# B&R Automation Studio project NAEUL004C00R13L518F00 (part 58)

#### Act_Background_TCPClose.st - Do Not Change!!!
```iecst
(** 2019-06-10 **)
ACTION Act_Background_TCPClose:

	//Close TCP Connection
	fbClose.udiTCPIdent	:= udiTCPIdent;
	fbClose(bEn := TRUE);

	IF fbClose.udiStatus = 0 THEN
		udiTCPIdent	:= 0;
		fbClose(bEn := FALSE);

		bRstConnection	:= FALSE;

	ELSIF fbClose.udiStatus < 65534 THEN
		udiTCPIdent	:= 0;
		eStatus1	:= Error;

		IF fbClose.udiStatus = 2300 THEN
			udiStatus1	:= 10027;	//Invalid Ident While Closing TCP
		ELSIF fbClose.udiStatus = 2310 THEN
			udiStatus1	:= 10028;	//Closing TCP Error
		ELSE
			udiStatus1	:= fbClose.udiStatus;
		END_IF

	END_IF

END_ACTION
```

#### Act_Background_Stop.st - Do Not Change!!!
```iecst
(** 2019-03-15 **)
ACTION Act_Background_Stop:

	IF bStop = TRUE THEN

		IF a_sMsgSend[0] = '' THEN

			bRstConnection	:= TRUE;

			IF udiTCPIdent = 0 THEN

				bRun	:= FALSE;

			END_IF

		END_IF

	END_IF

END_ACTION
```

#### Act_TCPSvr.st
```iecst
ACTION Act_TCPSvr:

	CASE usiStep OF
		0:
			//Analyse Connection
			IF udiSvrIdent = 0 THEN

				IF p_sSvrIP <> '' AND p_uiSvrPort <> 0 THEN
					usiStep	:= 1;
				END_IF

			ELSIF udiTCPIdent = 0 THEN

				usiStep	:= 2;

			END_IF

		1:
			//Create Server
			fbTCPSvrCreateSvr.sSvrIP				:= p_sSvrIP;
			fbTCPSvrCreateSvr.uiSvrPort				:= p_uiSvrPort;
			fbTCPSvrCreateSvr.udiAliveIdleTmInSec	:= 1;
			fbTCPSvrCreateSvr(bEn := TRUE);

			IF fbTCPSvrCreateSvr.udiStatus = 0 THEN
				udiSvrIdent	:= fbTCPSvrCreateSvr.udiTCPIdent;
				fbTCPSvrCreateSvr(bEn := FALSE);

				usiStep	:= 2;

			ELSIF fbTCPSvrCreateSvr.udiStatus < 65534 THEN
				fbTCPSvrCreateSvr(bEn := FALSE);

			END_IF

			IF p_bReconnect = TRUE THEN
				fbTCPSvrCreateSvr(bEn := FALSE);

				usiStep	:= 4;
			END_IF

		2:
			//Listen
			IF udiSvrIdent <> 0 THEN

				fbTCPSvrSvrListenFltr.bFltrIP			:= p_bFltrIP;
				fbTCPSvrSvrListenFltr.bFltrPort			:= p_bFltrPort;
				fbTCPSvrSvrListenFltr.a_sConfigIP[1]	:= p_sAllwClntIP;
				fbTCPSvrSvrListenFltr.a_uiConfigPort[1]	:= p_uiAllwClntPort;
				fbTCPSvrSvrListenFltr.udiSvrIdent		:= udiSvrIdent;
				fbTCPSvrSvrListenFltr(bEn := TRUE);

				IF fbTCPSvrSvrListenFltr.udiStatus = 0 THEN

					IF fbTCPSvrSvrListenFltr.bRejected = FALSE THEN
						udiTCPIdent	:= fbTCPSvrSvrListenFltr.udiClntIdent;
						fbTCPSvrSvrListenFltr(bEn := FALSE);
						bConnected		:= TRUE;

						usiStep	:= 3;
					ELSE
						fbTCPSvrSvrListenFltr(bEn := FALSE);
					END_IF

				ELSIF fbTCPSvrSvrListenFltr.udiStatus < 65534 THEN
					fbTCPSvrSvrListenFltr(bEn := FALSE);

				END_IF

			ELSE

				usiStep	:= 0;

			END_IF

			IF p_bReconnect = TRUE THEN
				fbTCPSvrSvrListenFltr(bEn := FALSE);

				usiStep	:= 4;
			END_IF

		3:
			//Send
			IF udiTCPIdent <> 0 AND bMsgSnd = TRUE THEN

				fbSend.udiTCPIdent	:= udiTCPIdent;
				fbSend.p_BffrDest	:= ADR(sMsgSnd);
				fbSend.udiSndSize	:= LEN(sMsgSnd);
				fbSend(bEn := TRUE);

				IF fbSend.udiStatus = 0 THEN
					bMsgSnd	:= FALSE;
					eSvrStat := SvrActIdle; //TCPSvrProcess
					fbSend(bEn := FALSE);

				ELSIF fbSend.udiStatus = 2320 THEN
					bMsgSnd	:= FALSE;
					fbSend(bEn := FALSE);

				ELSIF fbSend.udiStatus < 65534 THEN
					bMsgSnd	:= FALSE;
					fbSend(bEn := FALSE);

					usiStep	:= 4;

				END_IF

			ELSE
				fbSend(bEn := FALSE);

			END_IF

			//Receive
			IF udiTCPIdent <> 0 THEN

				fbRcv.udiTCPIdent	:= udiTCPIdent;
				fbRcv.p_BffrDest	:= ADR(sMsgRcv);
				fbRcv.udiBffrSize	:= SIZEOF(sMsgRcv);
				fbRcv(bEn := TRUE);

				IF eSvrStat <> SvrActWrite THEN
					eSvrStat := SvrActRead; //TCPSvrProcess
				END_IF

				IF fbRcv.udiStatus = 0 THEN
					bMsgRcv	:= TRUE;
					sSvrMsgRcv  := sMsgRcv;  //Evaluate
					fbRcv(bEn := FALSE);

				ELSIF fbRcv.udiStatus = 2316 THEN
					fbRcv(bEn := FALSE);

					usiStep	:= 4;

				ELSIF fbRcv.udiStatus = 2317 THEN //32605- no data is available for reading

					fbRcv(bEn := FALSE);
					memset(ADR(sMsgRcv) , 0 , SIZEOF(sMsgRcv));

				ELSIF fbRcv.udiStatus < 65534 THEN
					fbRcv(bEn := FALSE);

					usiStep	:= 4;

				END_IF

			ELSE
				fbRcv(bEn := FALSE);

			END_IF

			IF udiTCPIdent = 0 THEN
				usiStep	:= 0;
			END_IF

			IF p_bReconnect = TRUE THEN
				fbSend(bEn := FALSE);
				fbRcv(bEn := FALSE);

				usiStep	:= 4;
			END_IF

		4:
			//Close Client Ident
			IF udiTCPIdent <> 0 THEN

				fbClose.udiTCPIdent	:= udiTCPIdent;
				fbClose(bEn := TRUE);

				IF fbClose.udiStatus = 0 THEN
					udiTCPIdent	:= 0;
					fbClose(bEn := FALSE);
					bConnected		:= FALSE;

					usiStep	:= 5;

				ELSIF fbClose.udiStatus < 65534 THEN
					udiTCPIdent	:= 0;
					fbClose(bEn := FALSE);
					bConnected		:= FALSE;

				END_IF

			ELSE
				usiStep	:= 5;

			END_IF

		5:
			//Close Server Ident
			IF udiSvrIdent <> 0 THEN

				fbClose.udiTCPIdent	:= udiSvrIdent;
				fbClose(bEn := TRUE);

				IF fbClose.udiStatus = 0 THEN
					udiSvrIdent	:= 0;
					fbClose(bEn := FALSE);

					usiStep	:= 0;

				ELSIF fbClose.udiStatus < 65534 THEN
					udiSvrIdent	:= 0;
					fbClose(bEn := FALSE);

				END_IF

			ELSE
				usiStep	:= 0;

			END_IF

	END_CASE

END_ACTION
```

#### Act_TCPSvrProcess.st
```iecst
ACTION Act_TCPSvrProcess:

	CASE eSvrStat OF
		SvrActIdle:

		SvrActRead:
			//"Mag1Status","Mag2Status","Mag3Status","Mag4Status" >> 10:NA , 11:Error , 12:Ready, 13:Available ; 20:NA , 21:Error , 22:Ready, 23:Available

			eMagAGVStatus[0] := STRING_TO_USINT (LEFT(sSvrMsgRcv,FIND(sSvrMsgRcv, ',')-1));
			iSeparator 		:= FIND(sSvrMsgRcv, '$r$n');
			sData[0] := LEFT(sSvrMsgRcv, iSeparator-1);
			FOR i := 0 TO p_usiProjMag +(3 + 2*p_usiProjMag) DO 		//0:Dual ; 1:Triple; 2:Quar
				iSeparator := FIND(sData[i],',');
				IF iSeparator = 0 THEN
					;
				ELSE
					sData[i+1] := DELETE(sData[i],iSeparator+1,0);
				END_IF
			END_FOR

			IF bSingleMagLine THEN //single line magazine
				eMagAGVStatus[1] := STRING_TO_USINT (sData[1]);
			ELSE
				eMagAGVStatus[1] := STRING_TO_USINT (LEFT(sData[1],FIND(sData[1], ',')-1));
			END_IF

				eMagAGVStatus[2] := STRING_TO_USINT (LEFT(sData[2],FIND(sData[2], ',')-1));
			IF p_usiProjMag = 0 THEN//Dual mag
				eMagAGVStatus[3] := STRING_TO_USINT (sData[3]);
			ELSE //triple / quardrupal
				eMagAGVStatus[3] := STRING_TO_USINT (LEFT(sData[3],FIND(sData[3], ',')-1));
				eMagAGVStatus[4] := STRING_TO_USINT (LEFT(sData[4],FIND(sData[4], ',')-1));
				eMagAGVStatus[5] := STRING_TO_USINT (LEFT(sData[5],FIND(sData[5], ',')-1));
				eMagAGVStatus[6] := STRING_TO_USINT (LEFT(sData[6],FIND(sData[6], ',')-1));
				eMagAGVStatus[7] := STRING_TO_USINT (sData[7]);
			END_IF

			IF p_usiProjMag = 1 THEN//Triple mag
				eMagAGVStatus[5] := STRING_TO_USINT (sData[5]);
			ELSE
				eMagAGVStatus[5] := STRING_TO_USINT (LEFT(sData[5],FIND(sData[5], ',')-1));
				eMagAGVStatus[6] := STRING_TO_USINT (LEFT(sData[6],FIND(sData[6], ',')-1));
				eMagAGVStatus[7] := STRING_TO_USINT (sData[7]);
			END_IF

			IF eMagAGVStatus[0] >13 OR eMagAGVStatus[1] >12 OR eMagAGVStatus[2] >23 OR eMagAGVStatus[3] >22 OR
				eMagAGVStatus[4] >33 OR eMagAGVStatus[5] >32 OR eMagAGVStatus[6] >43 OR eMagAGVStatus[7] >42 OR

				eMagAGVStatus[0] <10 OR eMagAGVStatus[1] <10 OR eMagAGVStatus[2] <20 OR eMagAGVStatus[3] <20 OR
				eMagAGVStatus[4] <30 OR eMagAGVStatus[5] <30 OR eMagAGVStatus[6] <40 OR eMagAGVStatus[7] <40 THEN
				eSvrStatus := Error;
			END_IF

		SvrActRead1:
			//Structure: MagazineX, AGVStatus, AGVReq

			iSeparator 		:= FIND(sSvrMsgRcv, '$r$n');
			sData[0]		:= LEFT(sSvrMsgRcv, iSeparator-1); 		//magazine1 sData[0,1,2]
			sData[3] 		:= DELETE(sSvrMsgRcv,iSeparator+2,0);	//magazine2 sData[3,4,5]

			FOR i := 0 TO 5 DO
				iSeparator := FIND(sData[i],',');
				IF iSeparator = 0 THEN
					;
				ELSE
					sData[i+1] := DELETE(sData[i],iSeparator+1,0);
				END_IF
			END_FOR

			//check if endcode exist
			iSeparator := FIND(sData[i-1],'$r$n'); //where i = 6
			IF iSeparator = 0 THEN
				;
			ELSE
				sData[i-1] := DELETE(sData[i-1],iSeparator+1,iSeparator);
			END_IF

			tyAGVCurr[1].sAGVMag				:= LEFT(sData[0],FIND(sData[0], ',')-1);
			tyAGVCurr[1].eAGVStatus				:= STRING_TO_USINT (LEFT(sData[1],FIND(sData[1], ',')-1));
			tyAGVCurr[1].usiAGVReq				:= STRING_TO_USINT (sData[2]);
			tyAGVCurr[2].sAGVMag				:= LEFT(sData[3],FIND(sData[3], ',')-1);
			tyAGVCurr[2].eAGVStatus				:= STRING_TO_USINT (LEFT(sData[4],FIND(sData[4], ',')-1));
			tyAGVCurr[2].usiAGVReq				:= STRING_TO_USINT (sData[5]);

		SvrActWrite:
			//"Mag1Status","Mag2Status","Mag3Status","Mag4Status" >> 0:NA , 1:Error , 2:Ready, 3:Available
			//array [0][1]US1DS1 ,[2][3]US2DS2 ,[4][5]US3DS3, [6][7]US4DS4
			IF tyDTMagToAGV.bCI1Rdy  THEN
				a_sMagMcStatus[0] := '12'; //Ready, USB
			ELSE
				a_sMagMcStatus[0] := '10'; //NA
			END_IF
			IF tyDTMagToAGV.bCI1MagazineFull THEN
				a_sMagMcStatus[1] := '13'; //Available, DBA
			ELSE
				a_sMagMcStatus[1] := '10'; //NA
			END_IF;

			IF tyDTMagToAGV.bCI2Rdy  THEN
				a_sMagMcStatus[2] := '22';
			ELSE
				a_sMagMcStatus[2] := '20';
			END_IF;
			IF tyDTMagToAGV.bCI2MagazineFull THEN
				a_sMagMcStatus[3] := '23';
			ELSE
				a_sMagMcStatus[3] := '20';
			END_IF;

			IF tyDTMagToAGV.bCI3Rdy  THEN
				a_sMagMcStatus[4] := '32';
			ELSE
				a_sMagMcStatus[4] := '30';
			END_IF;
			IF tyDTMagToAGV.bCI3MagazineFull THEN
				a_sMagMcStatus[5] := '33';
			ELSE
				a_sMagMcStatus[5] := '30';
			END_IF;

			IF tyDTMagToAGV.bCI4Rdy  THEN
				a_sMagMcStatus[6] := '42';
			ELSE
				a_sMagMcStatus[6] := '40';
			END_IF;
			IF tyDTMagToAGV.bCI4MagazineFull THEN
				a_sMagMcStatus[7] := '43';
			ELSE
				a_sMagMcStatus[7] := '40';
			END_IF;
			//	sMsgSnd := USINT_TO_STRING (a_sMagMcStatus[3]);
			IF p_usiProjMag = 0 AND bSingleMagLine = FALSE THEN
				sMsgSnd := CONCAT(CONCAT(CONCAT(CONCAT(a_sMagMcStatus[0],','),CONCAT(a_sMagMcStatus[1],',')),CONCAT(a_sMagMcStatus[2],',')),CONCAT(a_sMagMcStatus[3],'$r$n'));
				bMsgSnd := TRUE;
			ELSIF bSingleMagLine THEN
				sMsgSnd := CONCAT(CONCAT(a_sMagMcStatus[0],','),CONCAT(a_sMagMcStatus[1],'$r$n'));
				bMsgSnd := TRUE;
			ELSE
				sMsgSnd := CONCAT(CONCAT(CONCAT(CONCAT(a_sMagMcStatus[0],','),CONCAT(a_sMagMcStatus[1],',')),CONCAT(a_sMagMcStatus[2],',')),a_sMagMcStatus[3]);
				sMsgSnd := CONCAT(CONCAT(CONCAT(CONCAT(CONCAT(sMsgSnd,','),CONCAT(a_sMagMcStatus[4],',')),CONCAT(a_sMagMcStatus[5],',')),CONCAT(a_sMagMcStatus[6],',')),CONCAT(a_sMagMcStatus[7],'$r$n'));
				bMsgSnd := TRUE;
			END_IF

	END_CASE;

	//Parse
	//Input (AGV to TCP(machine))
	bUBA 	:= eMagAGVStatus[0] = 13;
	bUBA2 	:= eMagAGVStatus[2] = 23;
	bDSB	:= eMagAGVStatus[1] = 12;
	bDSB2	:= eMagAGVStatus[3] = 22;

	//Output (Machine Sig(SOT) to TCP(AGV))
	tyDTMagToAGV.bCI1Rdy 			:= p_bUSB;
	tyDTMagToAGV.bCI1MagazineFull 	:= p_bDBA;
	tyDTMagToAGV.bCI2Rdy 			:= p_bUSB2;
	tyDTMagToAGV.bCI2MagazineFull 	:= p_bDBA2;

	fbTrig(CLK := p_bUSB);
	fbTrig1(CLK := p_bDBA);
	fbTrig2(CLK := p_bUSB2);
	fbTrig3(CLK := p_bDBA2);
	//	IF EDGEPOS(p_bUSB) OR EDGEPOS(p_bDBA) OR EDGEPOS(p_bUSB2) OR EDGEPOS(p_bDBA2)THEN
	IF fbTrig.Q OR fbTrig1.Q OR fbTrig2.Q OR fbTrig3.Q THEN
		eSvrStat := SvrActWrite;
	END_IF

END_ACTION
```

#### Act_Background_Log.st - Do Not Change!!!
```iecst
(** 2019-05-01 **)
ACTION Act_Background_Log:

	IF p_bLinkUIClearMsg THEN
		memset(ADR(a_tyHistoryList),0,SIZEOF(a_tyHistoryList));
		iHistoryCntr 	:= 1;
		p_bLinkUIClearMsg := FALSE;
	END_IF

	IF eStatus2 <> Error THEN

		IF udiWriteLogCntr <> udiLogCntr THEN

			CASE iWriteLogStep OF

				0:
					dtCurrDTTemp			:= p_dtCurrDT;
					fbFileAppend1.sFile		:= DT_TO_STRING(dtCurrDTTemp);
					fbFileAppend1.sFile		:= MID(fbFileAppend1.sFile , 10 , 4);
					fbFileAppend1.sFile		:= CONCAT('_' , fbFileAppend1.sFile);
					fbFileAppend1.sFile		:= CONCAT(p_sProgNm , fbFileAppend1.sFile);
					fbFileAppend1.sFile		:= CONCAT(fbFileAppend1.sFile , '.dat');

					fbFileAppend1.p_Src		:= ADR(a_sLogList[udiWriteLogCntr]);
					fbFileAppend1.udiLen	:= LEN(a_sLogList[udiWriteLogCntr]);

					iWriteLogStep	:= 1;

				1:
					fbFileAppend1(bEn := TRUE);
					IF fbFileAppend1.udiStatus = 0 THEN
						fbFileAppend1(bEn := FALSE);

						udiWriteLogCntr	:= udiWriteLogCntr + 1;
						IF udiWriteLogCntr = 11 THEN
							udiWriteLogCntr	:= 1;
						END_IF

						iWriteLogStep	:= 0;

					ELSIF fbFileAppend1.udiStatus < 65534 THEN
						eStatus2	:= Error;

						IF fbFileAppend1.udiStatus = 1900 THEN
							udiStatus2	:= 10018;	//File Open Error While Writing Log
						ELSIF fbFileAppend1.udiStatus = 1901 THEN
							udiStatus2	:= 10019;	//File Create Error While Writing Log
						ELSIF fbFileAppend1.udiStatus = 1913 THEN
							udiStatus2	:= 10020;	//Get File Info Error While Writing Log
						ELSIF fbFileAppend1.udiStatus = 1903 THEN
							udiStatus2	:= 10021;	//File Write Error While Writing Log
						ELSIF fbFileAppend1.udiStatus = 1904 THEN
							udiStatus2	:= 10022;	//File Close Error While Writing Log
						ELSIF fbFileAppend1.udiStatus = 1914 THEN
							udiStatus2	:= 10023;	//Directory Does Not Exist While Writing Log
						ELSE
							udiStatus2	:= fbFileAppend1.udiStatus;
						END_IF

						iWriteLogStep	:= 0;

					END_IF

			END_CASE

		END_IF

	END_IF

END_ACTION
```

#### Act_Main_Disable.st - Do Not Change!!!
```iecst
(** 2019-03-15 **)
ACTION Act_Main_Disable:

	bConnected		:= FALSE;

END_ACTION
```

#### InputRef.var - Do Not Change!!!
```iecst
(*2019-06-28*)
(**)
(*General*)
VAR
	p_bManual : REFERENCE TO BOOL;
	p_eAct : REFERENCE TO eTCPAction;
	p_udiRstErr : REFERENCE TO UDINT;
	p_bPrep : REFERENCE TO BOOL;
	p_bEn : REFERENCE TO BOOL;
	p_bDis : REFERENCE TO BOOL;
END_VAR
(**)
(*Configuration*)
VAR
	p_sSvrIP : REFERENCE TO STRING[15];
	p_uiSvrPort : REFERENCE TO UINT;
	p_uiClientPort : REFERENCE TO UINT;
	p_sMsgSnd : REFERENCE TO STRING[65535];
	p_sIPAddr : REFERENCE TO STRING[15];
	p_tyDTStructure : REFERENCE TO DTStructure;
	p_dtCurrDT : REFERENCE TO DATE_AND_TIME;
END_VAR
(*Listen Fltr*)
VAR
	p_eTCPModel : REFERENCE TO eTCPClientServer;
	p_bFltrIP : REFERENCE TO BOOL;
	p_bFltrPort : REFERENCE TO BOOL;
	p_sAllwClntIP : REFERENCE TO STRING[15];
	p_uiAllwClntPort : REFERENCE TO UINT;
	p_bReconnect : REFERENCE TO BOOL;
END_VAR
(**)
(*Input*)
VAR
	p_udiSndBffrSize : REFERENCE TO UDINT;
	p_udiRcvBffrSize : REFERENCE TO UDINT;
	p_udiAliveIdleTimeInSec : REFERENCE TO UDINT;
	p_tConnTimeOut : REFERENCE TO TIME;
	p_bOpsRun : REFERENCE TO BOOL;
	p_usiProjMag : REFERENCE TO USINT;
	p_sProgNm : REFERENCE TO STRING[15];
	p_bNtSettingsLoadDone : REFERENCE TO BOOL;
	p_udiFileKeepDay : REFERENCE TO UDINT;
END_VAR
(**)
VAR
	p_tyDTMagToAGV : REFERENCE TO tyTagDTMagToAGV;
END_VAR
(*Output from SOT to TCP*)
VAR
	p_bUSB : REFERENCE TO BOOL;
	p_bUSB2 : REFERENCE TO BOOL;
	p_bDBA : REFERENCE TO BOOL;
	p_bDBA2 : REFERENCE TO BOOL;
END_VAR
```

#### Act_Alarm.st - Do Not Change!!!
```iecst
(** 2019-03-25 **)
ACTION Act_Alarm:

	//Reset Error
	IF (eStatus = Error) AND bRstErr THEN
		p_eAct	:= TCPActIdle;
		eStat	:= TCPActIdle;
	END_IF

	IF p_udiRstErr <> udiRstErrOld THEN
		bRstErr			:= TRUE;
		udiRstErrOld	:= p_udiRstErr;
	ELSE
		bRstErr			:= FALSE;
	END_IF
	//Combine Error
	IF eStatus = Error OR eStatus1 = Error OR eStatus2 = Error THEN
		eMainStatus	:= Error;
	ELSE
		eMainStatus	:= eStatus;
	END_IF
	//Error
	IF EDGEPOS(eStatus = Error) THEN

		tyAlmData.sProgNm		:= p_sProgNm;
		tyAlmData.udiCode		:= udiStatus;
		tyAlmData.eSeverity		:= AlmSeverityError;
		tyAlmData.udiRunTime	:= tyAlmData.udiRunTime + 1;
		tyAlmData.bAlm			:= TRUE;
		tyAlmData.udiModuleNum  := udiModuleNum;
		g_sTCPProgNm		:= p_sProgNm;

		//Get Error Message
		IF tyAlmData.udiCode < 10000 OR tyAlmData.udiCode > 10199 THEN
			tyAlmData.sAlmMsg	:= 'Unknown';
			tyAlmData.sRcyMsg	:= 'Unknown';
		ELSE
			tyAlmData.sAlmMsg	:= a_tyAlmText[tyAlmData.udiCode].sAlmText;
			tyAlmData.sRcyMsg	:= a_tyAlmText[tyAlmData.udiCode].sRcyText;
		END_IF

		sStatTxt	:= tyAlmData.sAlmMsg;

	ELSIF bRstErr AND (tyAlmData.udiCode <> 0) THEN

		tyAlmData.udiCode	:= 0;
		tyAlmData.eSeverity	:= AlmSeverityNA;
		tyAlmData.sAlmMsg	:= '';
		tyAlmData.sRcyMsg	:= '';
		tyAlmData.bAlm			:= FALSE;
		sStatTxt	:= a_sStatText[eStat];

	END_IF

	//Error
	IF EDGEPOS(eStatus1 = Error) THEN

		tyAlmData1.sProgNm		:= p_sProgNm;
		tyAlmData1.udiCode		:= udiStatus1;
		tyAlmData1.eSeverity	:= AlmSeverityError;
		tyAlmData1.udiRunTime	:= tyAlmData1.udiRunTime + 1;
		tyAlmData1.bAlm			:= TRUE;
		tyAlmData1.udiModuleNum  := udiModuleNum;
		g_sTCPProgNm		:= p_sProgNm;

		//Get Error Message
		IF tyAlmData1.udiCode < 10000 OR tyAlmData1.udiCode > 10199 THEN
			tyAlmData1.sAlmMsg	:= 'Unknown';
			tyAlmData1.sRcyMsg	:= 'Unknown';
		ELSE
			tyAlmData1.sAlmMsg	:= a_tyAlmText[tyAlmData1.udiCode].sAlmText;
			tyAlmData1.sRcyMsg	:= a_tyAlmText[tyAlmData1.udiCode].sRcyText;
		END_IF

		sStatTxt	:= tyAlmData1.sAlmMsg;

	ELSIF bRstErr AND (tyAlmData1.udiCode <> 0) THEN

		tyAlmData1.udiCode		:= 0;
		tyAlmData1.eSeverity	:= AlmSeverityNA;
		tyAlmData1.sAlmMsg		:= '';
		tyAlmData1.sRcyMsg		:= '';
		tyAlmData1.bAlm			:= FALSE;
		sStatTxt	:= a_sStatText[eStat];

	END_IF

	//Error
	IF EDGEPOS(eStatus2 = Error) THEN

		tyAlmData2.sProgNm		:= p_sProgNm;
		tyAlmData2.udiCode		:= udiStatus2;
		tyAlmData2.eSeverity	:= AlmSeverityError;
		tyAlmData2.udiRunTime	:= tyAlmData2.udiRunTime + 1;
		tyAlmData2.bAlm			:= TRUE;
		tyAlmData2.udiModuleNum  := udiModuleNum;
		g_sTCPProgNm		:= p_sProgNm;

		//Get Error Message
		IF tyAlmData2.udiCode < 10000 OR tyAlmData2.udiCode > 10199 THEN
			tyAlmData2.sAlmMsg	:= 'Unknown';
			tyAlmData2.sRcyMsg	:= 'Unknown';
		ELSE
			tyAlmData2.sAlmMsg	:= a_tyAlmText[tyAlmData2.udiCode].sAlmText;
			tyAlmData2.sRcyMsg	:= a_tyAlmText[tyAlmData2.udiCode].sRcyText;
		END_IF

		sStatTxt	:= tyAlmData2.sAlmMsg;

	ELSIF bRstErr AND (tyAlmData2.udiCode <> 0) THEN

		tyAlmData2.udiCode		:= 0;
		tyAlmData2.eSeverity	:= AlmSeverityNA;
		tyAlmData2.sAlmMsg		:= '';
		tyAlmData2.sRcyMsg		:= '';
		tyAlmData2.bAlm			:= FALSE;
		sStatTxt	:= a_sStatText[eStat];

	END_IF

	//Error
	IF (bConnected = FALSE) THEN

		tyAlmData3.sProgNm		:= p_sProgNm;
		tyAlmData3.udiCode		:= udiStatus3;
		tyAlmData3.eSeverity	:= AlmSeverityWarning;
		tyAlmData3.udiRunTime	:= tyAlmData3.udiRunTime + 1;
		tyAlmData3.bWarning			:= TRUE;
		tyAlmData3.udiModuleNum  := udiModuleNum;
		g_sTCPProgNm		:= p_sProgNm;
		//Get Error Message
		IF tyAlmData3.udiCode < 10000 OR tyAlmData3.udiCode > 10199 THEN
			tyAlmData3.sAlmMsg	:= 'Unknown';
			tyAlmData3.sRcyMsg	:= 'Unknown';
		ELSE
			tyAlmData3.sAlmMsg	:= a_tyAlmText[tyAlmData3.udiCode].sAlmText;
			tyAlmData3.sRcyMsg	:= a_tyAlmText[tyAlmData3.udiCode].sRcyText;
			tyAlmData3.sRcyMsg	:= '';
		END_IF

		sStatTxt	:= tyAlmData3.sAlmMsg;

	ELSIF (bConnected AND (tyAlmData3.udiCode <> 0))  THEN

		tyAlmData3.udiCode		:= 0;
		tyAlmData3.eSeverity	:= AlmSeverityNA;
		tyAlmData3.sAlmMsg		:= '';
		tyAlmData3.sRcyMsg		:= '';
		tyAlmData3.bWarning		:= FALSE;
		sStatTxt	:= a_sStatText[eStat];

	END_IF
END_ACTION
```

#### Local.var - Do Not Change!!!
```iecst
(*2020-09-10*)
(**)
(*Local Action, State & Status*)
VAR
	bManual : BOOL := FALSE;
	eAct : eTCPAction := TCPActIdle;
	eStat : eTCPAction := TCPActIdle;
	eMainStatus : eFBStatus := Idle;
	eStatus : eFBStatus := Idle;
	eStatus1 : eFBStatus := Idle;
	eStatus2 : eFBStatus := Idle;
	udiStatus : UDINT := 0;
	udiStatus1 : UDINT := 0;
	udiStatus2 : UDINT := 0;
	udiStatus3 : UDINT := 0;
	udiStatus4 : UDINT := 0;
	udiStatus5 : UDINT := 0;
	sStatTxt : STRING[200] := '';
	a_sStatText : ARRAY[0..50] OF STRING[200] := ['Idling','Creating Directory','Deleting Old Log',48('')];
END_VAR
(**)
(*Local Alarm*)
VAR
	tyAlmData : tyAlmDat;
	tyAlmData1 : tyAlmDat;
	tyAlmData2 : tyAlmDat;
	tyAlmData3 : tyAlmDat;
	a_tyAlmText : ARRAY[10000..10199] OF tyAlmTxt := [(sAlmText:='Invalid Ident While Client Connecting',sRcyText:='Problem Occurred In The TCP/IP Connection. Check The Connection And Try To Reconnect.'),(sAlmText:='Setting Keep Alive Interval Time Error While Client Connecting',sRcyText:='Unable To Establish Connection Between Machine. Check For Setting And Resume Operation.'),(sAlmText:='Setting Keep Alive Idle Time Error While Client Connecting',sRcyText:='Unable To Establish Connection Between Machine. Check For Setting And Resume Operation.'),(sAlmText:='Setting Keep Alive Count Error While Client Connecting',sRcyText:='Unable To Establish Connection Between Machine. Check For Setting And Resume Operation.'),(sAlmText:='Setting Keep Alive Error While Client Connecting',sRcyText:='Unable To Establish Connection Between Machine. Check For Setting And Resume Operation.'),(sAlmText:='Setting Receive Buffer Error While Client Connecting',sRcyText:='Unable To Establish Connection Between Machine. Check For Setting And Resume Operation.'),(sAlmText:='Setting Send Buffer Error While Client Connecting',sRcyText:='Unable To Establish Connection Between Machine. Check For Setting And Resume Operation.'),(sAlmText:='Setting No Waiting Error While Client Connecting',sRcyText:='Unable To Establish Connection Between Machine. Check For Setting And Resume Operation.'),(sAlmText:='TCP Open Port Error While Client Connecting',sRcyText:='Problem Occurred In The TCP/IP Connection. Check The Connection And Try To Reconnect.'),(sAlmText:='Closing TCP Error While Client Connecting',sRcyText:='Problem Occurred In The TCP/IP Connection. Check The Connection And Try To Reconnect.'),(sAlmText:='Server Connection Failed While Client Connecting',sRcyText:='There Was A Problem Connecting To The Server. The Server May Not Exist or It is Unavailable At This Time. Check The Connection and Try Again.'),(sAlmText:='Ident In Used While Client Connecting',sRcyText:='Problem Occurred In The TCP/IP Connection. Check The Connection And Reconnect.'),(sAlmText:='TCP Connection Lost',sRcyText:='There Was A Problem Connecting To The Server. The Server May Not Exist or It is Unavailable At This Time. Check The Connection and Try Again.'),(sAlmText:='TCP Connection Lost',sRcyText:='Please Check Network Connection.'),(sAlmText:='Invalid Ident While Receiving Data',sRcyText:='Problem Occurred In The TCP/IP Connection. Check The Connection And Try To Reconnect.'),(sAlmText:='TCP Receive Data Error While Receiving Data',sRcyText:='Problem Occurred In The TCP/IP Connection. Check The Connection And Try To Reconnect.'),(sAlmText:='Create User Directory Error',sRcyText:='An Error Occurred While Attempting To Create User Directory. Please Contact Nutek For A Possible Solution'),(sAlmText:='Create Log Directory Error',sRcyText:='An Error Occurred While Attempting To Create User Directory. Please Contact Nutek For A Possible Solution'),(sAlmText:='File Open Error While Writing Log',sRcyText:='An Error Was Encountered While Trying To Open File. Please Contact Nutek For A Possible Solution.'),(sAlmText:='File Create Error While Writing Log',sRcyText:='An Error Was Encountered While Trying To Create File. Please Contact Nutek For A Possible Solution.'),(sAlmText:='Get File Info Error While Writing Log',sRcyText:='An Error Was Encountered While Getting File Info. Please Contact Nutek For A Possible Solution.'),(sAlmText:='File Write Error While Writing Log',sRcyText:='An Error Was Encountered While Getting File Info. Please Contact Nutek For A Possible Solution.'),(sAlmText:='File Close Error While Writing Log',sRcyText:='An Error Was Encountered While Trying To Close File. Please Contact Nutek For A Possible Solution.'),(sAlmText:='Directory Does Not Exist While Writing Log',sRcyText:='The Directory Does Not Exist.Please Contact Nutek For A Possible Solution.'),(sAlmText:='Invalid Ident While Sending Data',sRcyText:='Invalid Ident Value.'),(sAlmText:='TCP Retry Send Data Error While Sending Data',sRcyText:='Problem Occurred In The TCP/IP Connection. Check The Connection And Try To Reconnect.'),(sAlmText:='TCP Send Data Error',sRcyText:='Problem Occurred In The TCP/IP Connection. Check The Connection And Try To Reconnect.'),(sAlmText:='Invalid Ident While Closing TCP',sRcyText:='Invalid Ident Value.'),(sAlmText:='Closing TCP Error',sRcyText:='Problem Occurred In The TCP/IP Connection. Check The Connection And Try To Reconnect.'),171(0)];
END_VAR
(**)
(*Local Output*)
VAR
	bConnected : BOOL;
	bUSB : BOOL;
	bUBA : BOOL;
	bDSB : BOOL;
	bDBA : BOOL;
	bUSB2 : BOOL;
	bUBA2 : BOOL;
	bDSB2 : BOOL;
	bDBA2 : BOOL;
END_VAR
(**)
(*Local Input*)
VAR
	sSvrIP : STRING[15] := '192.168.0.16';
	uiSvrPort : UINT := 7171;
	uiClientPort : UINT := 5000;
	udiRstErr : UDINT := 0;
	bPrep : BOOL := TRUE;
	bEn : BOOL := TRUE;
	bDis : BOOL := FALSE;
	sIPAddr : STRING[15] := '192.168.0.16';
	tyDTStructure : DTStructure := (year:=2019,month:=01,day:=05,wday:=05,hour:=21,minute:=28,second:=30,millisec:=123,microsec:=456);
	dtCurrDT : DATE_AND_TIME := DT#2019-02-23-12:30:50;
	udiSndBffrSize : UDINT := 65536;
	udiRcvBffrSize : UDINT := 65536;
	udiAliveIdleTimeInSec : UDINT := 5;
	tConnTimeOut : TIME := T#30s;
	bOpsRun : BOOL := FALSE;
	udiFileKeepDay : UDINT := 30;
	usiProjMag : USINT := 0;
	sProgNm : STRING[15] := 'TCP';
	bNtSettingsLoadDone : BOOL := TRUE;
END_VAR
(**)
(*Local*)
VAR
	eTCPModel : eTCPClientServer := Server;
	eStatOld : eTCPAction := TCPActIdle;
	bRstErr : BOOL;
	udiRstErrOld : UDINT;
	bInitDone : BOOL;
	bInitialDone : BOOL;
	bRun : BOOL;
	bStop : BOOL;
	bRstConnection : BOOL;
	bRstState : BOOL;
	usiStep : USINT;
	udiTCPIdent : UDINT; (*Client ident*)
	udiMsgSendBffr : UDINT;
	udiSndMsgLen : UDINT;
	iFindBatteryLvl : INT;
	rCurrentBatteryLvl : REAL;
	sExtractBatteryLvl : STRING[30];
	sDecodeMsg : STRING[65535];
	a_sMsgSend : ARRAY[0..50] OF STRING[65535];
	bMsgSnd : BOOL;
	bMsgRcv : BOOL;
	sMsgSnd : STRING[65535];
	sMsgRcv : STRING[65535];
	sSvrMsgRcv : STRING[65535];
	sSnd : STRING[65535];
	sRcv : STRING[65535];
	fbClntConnect : fbTCPClntConnect;
	fbTCPSvrCreateSvr : fbTCPCreateSvr;
	fbTCPSvrSvrListenFltr : fbTCPSvrListenFltr;
	fbRcv : fbTCPRcv;
	fbSend : fbTCPSnd;
	fbClose : fbTCPClose;
	fbTrig : RF_TRIG;
	fbTrig1 : RF_TRIG;
	fbTrig2 : RF_TRIG;
	fbTrig3 : RF_TRIG;
	udiLogCntr : UDINT := 1;
	udiWriteLogCntr : UDINT := 1;
	a_sLogList : ARRAY[1..10] OF STRING[65535];
	sDT : STRING[80];
	dtCurrDTTemp : DATE_AND_TIME;
	fbDirCreate1 : fbDirCreate;
	fbDirCreate2 : fbDirCreate;
	fbFileAppend1 : fbFileFullAppend;
	fbFileOldDel1 : fbFileOldDel;
	iWriteLogStep : INT := 0;
	iHistoryCntr : INT := 1;
	a_tyHistoryList : ARRAY[1..8] OF tyTCPHistoryMsg;
	bLoginSuccess : BOOL;
	bCheckAliveTimeout : BOOL;
	bWaitAliveResponse : BOOL;
	fbSendAliveTimer : TON;
	fbCheckAliveTimer : TON;
END_VAR
(**)
VAR
	tyAIVMsgRcvData : tyAIVMsgRcvDat;
	sELD1Reached : STRING[80] := 'Arrived At ELD1';
	sELD1Completed : STRING[80] := 'ELD1_completed';
	sELD2Reached : STRING[80] := 'Arrived At ELD2';
	sELD2Completed : STRING[80] := 'ELD2_completed';
	sELD3Reached : STRING[80] := 'Arrived At ELD3';
	sELD3Completed : STRING[80] := 'ELD3_completed';
	sEUL1Reached : STRING[80] := 'Arrived At EUL1';
	sEUL1Completed : STRING[80] := 'EUL1_completed';
	sEUL2Reached : STRING[80] := 'Arrived At EUL2';
	sEUL2Completed : STRING[80] := 'EUL2_completed';
	sEUL3Reached : STRING[80] := 'Arrived At EUL3';
	sEUL3Completed : STRING[80] := 'EUL3_completed';
	sSTANDBYReached : STRING[80] := 'Arrived At STANDBY';
	sSTANDBYCompleted : STRING[80] := 'STANDBY_completed';
END_VAR
(*Server*)
VAR
	udiSvrIdent : UDINT := 0;
	bFltrIP : BOOL;
	bFltrPort : BOOL;
	sAllwClntIP : STRING[15];
	uiAllwClntPort : UINT;
	bReconnect : BOOL;
	eSvrStat : eTCPSvrAction := SvrActIdle;
	eSvrStatus : eFBStatus := Idle;
	bSingleMagLine : BOOL := FALSE;
END_VAR
(**)
(*Data Parameter(Read1)*)
VAR
	i : INT;
	iSeparator : INT := 0;
	tyAGVCurr : ARRAY[1..2] OF tyTCPAGVDetail;
	sData : ARRAY[0..7] OF STRING[30]; (*Buffer *)
END_VAR
(*Data Parameter(Read/write)*)
VAR
	eMagAGVStatus : ARRAY[0..7] OF eTCPAGVStatus := [8(AGVNA)];
	a_sMagMcStatus : ARRAY[0..7] OF STRING[2] := [8('')];
	tyDTMagToAGV : tyTagDTMagToAGV;
	udiModuleNum : UDINT := 4301;
END_VAR
```

#### Act_Action.st - not listed in the package file held
```iecst
(** 2019-03-25 **)
ACTION Act_Action:

//Reset Error
	IF (eStatus = Error) AND bRstErr THEN
		p_eAct	:= TCPActIdle;
		eStat	:= TCPActIdle;
	END_IF

	//Set p_eAct
	IF eStatus = Idle OR eStatus = Busy OR eStatus = Done THEN
		eStat	:= p_eAct;
	END_IF

END_ACTION
```

#### Act_Alarm1.st - not listed in the package file held
```iecst
(** 2019-03-25 **)
ACTION Act_Alarm1:

	//Error
	IF EDGEPOS(eStatus1 = Error) THEN

		tyAlmData1.sProgNm		:= p_sProgNm;
		tyAlmData1.udiCode		:= udiStatus1;
		tyAlmData1.eSeverity	:= AlmSeverityError;
		tyAlmData1.udiRunTime	:= tyAlmData1.udiRunTime + 1;
		tyAlmData1.bAlm			:= TRUE;
		tyAlmData1.udiModuleNum  := udiModuleNum;
		g_sTCPProgNm		:= p_sProgNm;

		//Get Error Message
		IF tyAlmData1.udiCode < 10000 OR tyAlmData1.udiCode > 10199 THEN
			tyAlmData1.sAlmMsg	:= 'Unknown';
			tyAlmData1.sRcyMsg	:= 'Unknown';
		ELSE
			tyAlmData1.sAlmMsg	:= a_tyAlmText[tyAlmData1.udiCode].sAlmText;
			tyAlmData1.sRcyMsg	:= a_tyAlmText[tyAlmData1.udiCode].sRcyText;
		END_IF

		sStatTxt	:= tyAlmData1.sAlmMsg;

	ELSIF bRstErr AND (tyAlmData1.udiCode <> 0) THEN

		tyAlmData1.udiCode		:= 0;
		tyAlmData1.eSeverity	:= AlmSeverityNA;
		tyAlmData1.sAlmMsg		:= '';
		tyAlmData1.sRcyMsg		:= '';
		tyAlmData1.bAlm			:= FALSE;
		sStatTxt	:= a_sStatText[eStat];

	END_IF

END_ACTION
```

#### Act_Alarm2.st - not listed in the package file held
```iecst
(** 2019-03-25 **)
ACTION Act_Alarm2:

	//Error
	IF EDGEPOS(eStatus2 = Error) THEN

		tyAlmData2.sProgNm		:= p_sProgNm;
		tyAlmData2.udiCode		:= udiStatus2;
		tyAlmData2.eSeverity	:= AlmSeverityError;
		tyAlmData2.udiRunTime	:= tyAlmData2.udiRunTime + 1;
		tyAlmData2.bAlm			:= TRUE;
		tyAlmData2.udiModuleNum  := udiModuleNum;
		g_sTCPProgNm		:= p_sProgNm;

		//Get Error Message
		IF tyAlmData2.udiCode < 10000 OR tyAlmData2.udiCode > 10199 THEN
			tyAlmData2.sAlmMsg	:= 'Unknown';
			tyAlmData2.sRcyMsg	:= 'Unknown';
		ELSE
			tyAlmData2.sAlmMsg	:= a_tyAlmText[tyAlmData2.udiCode].sAlmText;
			tyAlmData2.sRcyMsg	:= a_tyAlmText[tyAlmData2.udiCode].sRcyText;
		END_IF

		sStatTxt	:= tyAlmData2.sAlmMsg;

	ELSIF bRstErr AND (tyAlmData2.udiCode <> 0) THEN

		tyAlmData2.udiCode		:= 0;
		tyAlmData2.eSeverity	:= AlmSeverityNA;
		tyAlmData2.sAlmMsg		:= '';
		tyAlmData2.sRcyMsg		:= '';
		tyAlmData2.bAlm			:= FALSE;
		sStatTxt	:= a_sStatText[eStat];

	END_IF

END_ACTION
```

#### Act_Alarm3.st - not listed in the package file held
```iecst
(** 2020-09-10 **)
ACTION Act_Alarm3:

	//Error
	IF (bConnected = FALSE) THEN

		tyAlmData3.sProgNm		:= p_sProgNm;
		tyAlmData3.udiCode		:= udiStatus3;
		tyAlmData3.eSeverity	:= AlmSeverityWarning;
		tyAlmData3.udiRunTime	:= tyAlmData3.udiRunTime + 1;
		tyAlmData3.bWarning			:= TRUE;
		tyAlmData3.udiModuleNum  := udiModuleNum;
		g_sTCPProgNm		:= p_sProgNm;
		//Get Error Message
		IF tyAlmData3.udiCode < 10000 OR tyAlmData3.udiCode > 10199 THEN
			tyAlmData3.sAlmMsg	:= 'Unknown';
			tyAlmData3.sRcyMsg	:= 'Unknown';
		ELSE
			tyAlmData3.sAlmMsg	:= a_tyAlmText[tyAlmData3.udiCode].sAlmText;
			tyAlmData3.sRcyMsg	:= a_tyAlmText[tyAlmData3.udiCode].sRcyText;
			tyAlmData3.sRcyMsg	:= '';
		END_IF

		sStatTxt	:= tyAlmData3.sAlmMsg;

	ELSIF (bConnected AND (tyAlmData3.udiCode <> 0))  THEN

		tyAlmData3.udiCode		:= 0;
		tyAlmData3.eSeverity	:= AlmSeverityNA;
		tyAlmData3.sAlmMsg		:= '';
		tyAlmData3.sRcyMsg		:= '';
		tyAlmData3.bWarning		:= FALSE;
		sStatTxt	:= a_sStatText[eStat];

	END_IF

END_ACTION
```

#### Act_CombineErr.st - not listed in the package file held
```iecst
(** 2019-03-15 **)
ACTION Act_CombineErr:

	//Combine Error
	IF eStatus = Error OR eStatus1 = Error OR eStatus2 = Error THEN
		eMainStatus	:= Error;
	ELSE
		eMainStatus	:= eStatus;
	END_IF

END_ACTION
```

#### Act_InitGlobal.st - not listed in the package file held
```iecst
(** 2019-06-28 **)
ACTION Act_InitGlobal:

	(* Always Change If Project Change *)

	//Pass Data To Link
//	p_bLinkStartupRun ACCESS p_StartupRun;
//	p_bLinkUIClearMsg ACCESS p_UITCPClearMsg;
//	p_bLinkConnectEn ACCESS p_UITCPConnectionEn;
	p_bUSB ACCESS p_USSOT1USB;
	p_bUSB2 ACCESS p_USSOT2USB;
	p_bDBA ACCESS p_DSSOT1DBA;
	p_bDBA2 ACCESS p_DSSOT2DBA;
	p_eLinkAGVComProtocol ACCESS p_McParamAGVComProtocol;

	//Pass Data To Internal Use
//	p_bManual ACCESS p_UIUIMnlMod;
	p_udiRstErr ACCESS p_RstErrReset;
	p_sIPAddr ACCESS p_HWInfoIPAddr;
	p_tyDTStructure ACCESS p_TimeCurrDTStruct;
	p_dtCurrDT ACCESS p_TimeCurrDT;
	p_bOpsRun ACCESS p_OpsRun;
	p_sMsgSnd ACCESS ADR(sMsgSnd);
	p_sSvrIP ACCESS p_HWInfoIPAddr;
	p_uiSvrPort ACCESS p_McParamTCPSvrPort; //UI setting input

	p_usiProjMag ACCESS p_NtParamProjMag;

	p_bNtSettingsLoadDone ACCESS p_StartupNtSettingsLoadDone;

	(* Always Change If Project Change *)

END_ACTION
```

#### Init.st - not listed in the package file held
```iecst
(** 2020-09-10 **)
PROGRAM _INIT

	(* Always Change If Project Change *)

	//Pass Address To Global Address For External Use
	//Action, State & Status
	p_TCPStat		:= ADR(eStat);
	p_TCPStatus		:= ADR(eMainStatus);
	p_TCPStatTxt	:= ADR(sStatTxt);

	//Alarm
	p_TCPAlmData	:= ADR(tyAlmData);
	p_TCPAlmData1	:= ADR(tyAlmData1);
	p_TCPAlmData2	:= ADR(tyAlmData2);
	p_TCPAlmData3	:= ADR(tyAlmData3);

	//Output
	p_TCPConnected				:= ADR(bConnected);
	p_TCPHistoryList			:= ADR(a_tyHistoryList);
	p_TCPAIVBatteryLvl			:= ADR(sExtractBatteryLvl);
	p_TCPAIVCurrentBatteryLvl	:= ADR(rCurrentBatteryLvl);
	p_TCPMsgRcvData				:= ADR(tyAIVMsgRcvData); //Client

	p_TCPSvrMsgRcvData			:= ADR(sSvrMsgRcv);
	p_TCPSvrAGVStatus1			:= ADR(eMagAGVStatus[0]);
	p_TCPSvrAGVStatus2			:= ADR(eMagAGVStatus[1]);
	p_TCPSvrAGVStatus3			:= ADR(eMagAGVStatus[2]);
	p_TCPSvrAGVStatus4			:= ADR(eMagAGVStatus[3]);

	p_TCPSvrUBA					:= ADR(bUBA);
	p_TCPSvrUBA2				:= ADR(bUBA2);
	p_TCPSvrDSB					:= ADR(bDSB);
	p_TCPSvrDSB2				:= ADR(bDSB2);
	(* Always Change If Project Change *)

END_PROGRAM
```

### TCPTop.var - Change By Project
```iecst
(*2019-06-02*)
(**)
(*Constant*)
(**)
(*Action & State & Status*)
VAR
	p_TCPTopStat : UDINT;
	p_TCPTopStatus : UDINT;
	p_TCPTopStatTxt : UDINT;
END_VAR
(**)
(*Alarm*)
VAR
	p_TCPTopAlmData : UDINT;
END_VAR
(**)
(*Output*)
VAR
	p_TCPTopFullMsgRd : UDINT;
	p_TCPTopMsgRd : UDINT;
	p_TCPTopMsgRdValid : UDINT;
	p_TCPTopMsgRdLen : UDINT;
END_VAR
```

### Program Logical/TCP/TCPTop (IEC) - 1.00.0 - NtRecipe v5.00.0 , NtFileIO v5.00.0

#### InputRef.var
```iecst
(*2019-06-07*)
(**)
(*General*)
VAR
	p_eAct : REFERENCE TO eTCPAction1;
	p_udiRstErr : REFERENCE TO UDINT;
	p_bPrep : REFERENCE TO BOOL;
	p_bEn : REFERENCE TO BOOL;
	p_bDis : REFERENCE TO BOOL;
	p_bRun : REFERENCE TO BOOL;
END_VAR
(**)
(*Configuration*)
VAR
	p_sClntIP : REFERENCE TO STRING[15];
	p_sSvrIP : REFERENCE TO STRING[15];
	p_uiClntPort : REFERENCE TO UINT;
	p_uiSvrPort : REFERENCE TO UINT;
	p_udiSndBffrSize : REFERENCE TO UDINT;
	p_udiRcvBffrSize : REFERENCE TO UDINT;
	p_udiAliveIdleTmInSec : REFERENCE TO UDINT;
	p_tConnectTO : REFERENCE TO TIME;
	p_sMsgWr : REFERENCE TO STRING[80];
	p_diStartCode1 : REFERENCE TO DINT;
	p_diStartCode2 : REFERENCE TO DINT;
	p_diEndCode1 : REFERENCE TO DINT;
	p_diEndCode2 : REFERENCE TO DINT;
	p_sProgNm : REFERENCE TO STRING[15];
	p_bNtSettingsLoadDone : REFERENCE TO BOOL;
	p_usiTravLifScanCntr : REFERENCE TO USINT;
END_VAR
```

#### Local.var
```iecst
(*2019-06-07*)
(**)
(*Local Action, State & Status*)
VAR
	eAct : eTCPAction1 := TCPActIdle_0;
	eStat : eTCPAction1 := TCPActIdle_0;
	eStatus : eFBStatus := Idle;
	udiStatus : UDINT := 0;
	sStatTxt : STRING[200] := '';
	a_sStatText : ARRAY[0..50] OF STRING[200] := ['Idling','TCP Write Then Read','TCP Write Then Read Until Valid',48('')];
END_VAR
(**)
(*Local Alarm*)
VAR
	tyAlmData : tyAlmDat;
	a_tyAlmText : ARRAY[10000..10099] OF tyAlmTxt := [(sAlmText:='TCP Open Port Error While Full Write & Read',sRcyText:='Pleae Contact Nutek For Future Possible Solution'),(sAlmText:='Invalid Ident While Full Write & Read',sRcyText:='Pleae Contact Nutek For Future Possible Solution'),(sAlmText:='Setting Send Buffer Error While Full Write & Read',sRcyText:='Pleae Contact Nutek For Future Possible Solution'),(sAlmText:='Setting Receive Buffer Error While Full Write & Read',sRcyText:='Pleae Contact Nutek For Future Possible Solution'),(sAlmText:='Setting No Waiting Error While Full Write & Read',sRcyText:='Pleae Contact Nutek For Future Possible Solution'),(sAlmText:='Setting Keep Alive Error While Full Write & Read',sRcyText:='Pleae Contact Nutek For Future Possible Solution'),(sAlmText:='Setting Keep Alive Count Error While Full Write & Read',sRcyText:='Pleae Contact Nutek For Future Possible Solution'),(sAlmText:='Setting Keep Alive Idle Time Error While Full Write & Read',sRcyText:='Pleae Contact Nutek For Future Possible Solution'),(sAlmText:='Setting Keep Alive Interval Time Error While Full Write & Read',sRcyText:='Pleae Contact Nutek For Future Possible Solution'),(sAlmText:='Server Connection Failed While Full Write & Read',sRcyText:='Check Whether Server Connection Is Valid'),(sAlmText:='Ident In Used While Full Write & Read',sRcyText:='Pleae Contact Nutek For Future Possible Solution'),(sAlmText:='Connect To Server Error While Full Write & Read',sRcyText:='Check Whether Server Connection Is Valid'),(sAlmText:='Client Connect Time Out While Full Write & Read',sRcyText:='Check Whether Server Connection Is Valid'),(sAlmText:='Closing TCP Error While Full Write & Read',sRcyText:='Pleae Contact Nutek For Future Possible Solution'),(sAlmText:='TCP Retry Send Data Error While Full Write & Read',sRcyText:='Pleae Contact Nutek For Future Possible Solution'),(sAlmText:='Invalid Ident While Full Write & Read',sRcyText:='Pleae Contact Nutek For Future Possible Solution'),(sAlmText:='Opposite Closed Connection While Full Write & Read',sRcyText:='Check Whether Server Connection Is Valid'),(sAlmText:='TCP Send Data Error While Full Write & Read',sRcyText:='Pleae Contact Nutek For Future Possible Solution'),(sAlmText:='Data Receive Length Is Zero Due To Opposite Closed Connection While TCP Receiving Data While Full Write & Read',sRcyText:='Check Whether Server Connection Is Valid'),(sAlmText:='Invalid Ident While Full Write & Read',sRcyText:='Pleae Contact Nutek For Future Possible Solution'),(sAlmText:='Opposite Closed Connection While Full Write & Read',sRcyText:='Check Whether Server Connection Is Valid'),(sAlmText:='TCP Receive Data Error While Full Write & Read',sRcyText:='Pleae Contact Nutek For Future Possible Solution'),(sAlmText:='Invalid Ident While Full Write & Read',sRcyText:='Pleae Contact Nutek For Future Possible Solution'),(sAlmText:='Closing TCP Error While Full Write & Read',sRcyText:='Pleae Contact Nutek For Future Possible Solution'),(sAlmText:='TCP Open Port Error While Full Write & Read Until Valid',sRcyText:='Pleae Contact Nutek For Future Possible Solution'),(sAlmText:='Invalid Ident While Full Write & Read Until Valid',sRcyText:='Pleae Contact Nutek For Future Possible Solution'),(sAlmText:='Setting Send Buffer Error While Full Write & Read Until Valid',sRcyText:='Pleae Contact Nutek For Future Possible Solution'),(sAlmText:='Setting Receive Buffer Error While Full Write & Read Until Valid',sRcyText:='Pleae Contact Nutek For Future Possible Solution'),(sAlmText:='Setting No Waiting Error While Full Write & Read Until Valid',sRcyText:='Pleae Contact Nutek For Future Possible Solution'),(sAlmText:='Setting Keep Alive Error While Full Write & Read Until Valid',sRcyText:='Pleae Contact Nutek For Future Possible Solution'),(sAlmText:='Setting Keep Alive Count Error While Full Write & Read Until Valid',sRcyText:='Pleae Contact Nutek For Future Possible Solution'),(sAlmText:='Setting Keep Alive Idle Time Error While Full Write & Read Until Valid',sRcyText:='Pleae Contact Nutek For Future Possible Solution'),(sAlmText:='Setting Keep Alive Interval Time Error While Full Write & Read Until Valid',sRcyText:='Pleae Contact Nutek For Future Possible Solution'),(sAlmText:='Server Connection Failed While Full Write & Read Until Valid',sRcyText:='Check Whether Server Connection Is Valid'),(sAlmText:='Ident In Used While Full Write & Read Until Valid',sRcyText:='Pleae Contact Nutek For Future Possible Solution'),(sAlmText:='Connect To Server Error While Full Write & Read Until Valid',sRcyText:='Check Whether Server Connection Is Valid'),(sAlmText:='Client Connect Time Out While Full Write & Read Until Valid',sRcyText:='Check Whether Server Connection Is Valid'),(sAlmText:='Closing TCP Error While Full Write & Read Until Valid',sRcyText:='Pleae Contact Nutek For Future Possible Solution'),(sAlmText:='TCP Retry Send Data Error While Full Write & Read Until Valid',sRcyText:='Pleae Contact Nutek For Future Possible Solution'),(sAlmText:='Invalid Ident While Full Write & Read Until Valid',sRcyText:='Pleae Contact Nutek For Future Possible Solution'),(sAlmText:='Opposite Closed Connection While Full Write & Read Until Valid',sRcyText:='Check Whether Server Connection Is Valid'),(sAlmText:='TCP Send Data Error While Full Write & Read Until Valid',sRcyText:='Pleae Contact Nutek For Future Possible Solution'),(sAlmText:='Data Receive Length Is Zero Due To Opposite Closed Connection While TCP Receiving Data While Full Write & Read Until Valid',sRcyText:='Check Whether Server Connection Is Valid'),(sAlmText:='Invalid Ident While Full Write & Read Until Valid',sRcyText:='Pleae Contact Nutek For Future Possible Solution'),(sAlmText:='Opposite Closed Connection While Full Write & Read Until Valid',sRcyText:='Check Whether Server Connection Is Valid'),(sAlmText:='TCP Receive Data Error While Full Write & Read Until Valid',sRcyText:='Pleae Contact Nutek For Future Possible Solution'),(sAlmText:='Invalid Ident While Full Write & Read Until Valid',sRcyText:='Pleae Contact Nutek For Future Possible Solution'),(sAlmText:='Closing TCP Error While Full Write & Read Until Valid',sRcyText:='Pleae Contact Nutek For Future Possible Solution'),52(0)];
END_VAR
(**)
(*Local Output*)
VAR
	sFullMsgRd : STRING[80];
	sMsgRd : STRING[80];
	bMsgRdValid : BOOL;
	uiMsgRdLen : UINT;
END_VAR
(**)
(*Local Input*)
VAR
	udiRstErr : UDINT := 0;
	bPrep : BOOL := TRUE;
	bEn : BOOL := TRUE;
	bDis : BOOL := FALSE;
	bRun : BOOL := FALSE;
	sClntIP : STRING[15];
	sSvrIP : STRING[15];
	uiClntPort : UINT;
	uiSvrPort : UINT;
	udiSndBffrSize : UDINT := 65536;
	udiRcvBffrSize : UDINT := 65536;
	udiAliveIdleTmInSec : UDINT := 10;
	tConnectTO : TIME := T#30s;
	sMsgWr : STRING[80] := 'T'; (*trigger scanner*)
	diStartCode1 : DINT := -1;
	diStartCode2 : DINT := -1;
	diEndCode1 : DINT := -1;
	diEndCode2 : DINT := -1;
	sProgNm : STRING[15] := 'TCPTop';
	bNtSettingsLoadDone : BOOL := TRUE;
END_VAR
(**)
(*Local*)
VAR
	bRstErr : BOOL;
	udiRstErrOld : UDINT;
	bInitDone : BOOL;
	bInitialDone : BOOL;
	fbClntConnect : fbTCPClntConnect;
	fbSnd : fbTCPSnd;
	fbRcv : fbTCPRcv;
	fbClose : fbTCPClose;
	udiTCPIdent : UDINT;
	udiTCPIdent1 : UDINT;
	usiStep : USINT;
	iStartCodeLen : INT;
	siStartCode1 : SINT;
	siStartCode2 : SINT;
	sStartCode : STRING[2];
	iStartCodePos : INT;
	iEndCodeLen : INT;
	siEndCode1 : SINT;
	siEndCode2 : SINT;
	sEndCode : STRING[2];
	iEndCodePos : INT;
	bRstConnection : BOOL;
	usiScanCntr : USINT;
END_VAR
```

#### Act_Action.st
```iecst
(** 2019-06-02 **)
ACTION Act_Action:

	//Reset Error
	IF (eStatus = Error) AND bRstErr THEN
		p_eAct	:= TCPActIdle_0;
		eStat	:= TCPActIdle_0;
	END_IF

	//Set p_eAct
	IF eStatus = Idle OR eStatus = Busy OR eStatus = Done THEN
		eStat	:= p_eAct;
	END_IF

END_ACTION
```

#### Act_Alarm.st
```iecst
(** 2019-06-02 **)
ACTION Act_Alarm:

	//Error
	IF EDGEPOS(eStatus = Error) THEN

		tyAlmData.sProgNm		:= p_sProgNm;
		tyAlmData.udiCode		:= udiStatus;
		tyAlmData.eSeverity		:= AlmSeverityError;
		tyAlmData.udiRunTime	:= tyAlmData.udiRunTime + 1;

		//Get Error Message
		IF tyAlmData.udiCode < 10000 OR tyAlmData.udiCode > 10099 THEN
			tyAlmData.sAlmMsg	:= 'Unknown';
			tyAlmData.sRcyMsg	:= 'Unknown';
		ELSE
			tyAlmData.sAlmMsg	:= a_tyAlmText[tyAlmData.udiCode].sAlmText;
			tyAlmData.sRcyMsg	:= a_tyAlmText[tyAlmData.udiCode].sRcyText;
		END_IF

		sStatTxt	:= tyAlmData.sAlmMsg;

	ELSIF bRstErr AND (tyAlmData.udiCode <> 0) THEN

		tyAlmData.udiCode	:= 0;
		tyAlmData.eSeverity	:= AlmSeverityNA;
		tyAlmData.sAlmMsg	:= '';
		tyAlmData.sRcyMsg	:= '';

		sStatTxt	:= a_sStatText[eStat];

	END_IF

END_ACTION
```

#### Act_InitGlobal.st
```iecst
(** 2019-06-02 **)
ACTION Act_InitGlobal:

	(* Always Change If Project Change *)

	//Pass Data To Link

	//Pass Data To Internal Use
	p_bPrep ACCESS p_NtParamProjScanPrep;
	p_bEn ACCESS p_McParamTopScannerEn;
	p_udiRstErr ACCESS p_RstErrReset;

	p_sClntIP ACCESS p_HWInfoIPAddr;
	p_sSvrIP ACCESS p_McParamTopScanIP;
	p_uiSvrPort ACCESS p_McParamTopScanPort;
	p_bRun ACCESS p_OpsRun;

	p_bNtSettingsLoadDone ACCESS p_StartupNtSettingsLoadDone;
	p_usiTravLifScanCntr ACCESS p_OpsTravLifScanCntr;
	(* Always Change If Project Change *)

END_ACTION
```

#### Act_InitLocal.st
```iecst
(** 2019-06-07 **)
ACTION Act_InitLocal:

	//Input Reference Link To Local Variable
	p_eAct ACCESS ADR(eAct);
	p_udiRstErr ACCESS ADR(udiRstErr);
	p_bPrep ACCESS ADR(bPrep);
	p_bEn ACCESS ADR(bEn);
	p_bDis ACCESS ADR(bDis);

	p_sClntIP ACCESS ADR(sClntIP); //plc ip
	p_sSvrIP ACCESS ADR(sSvrIP); //scanner ip
	p_uiClntPort ACCESS ADR(uiClntPort); //def :0
	p_uiSvrPort ACCESS ADR(uiSvrPort); //scanner port
	p_bRun ACCESS ADR(bRun); ;
	p_udiSndBffrSize ACCESS ADR(udiSndBffrSize);
	p_udiRcvBffrSize ACCESS ADR(udiRcvBffrSize);
	p_udiAliveIdleTmInSec ACCESS ADR(udiAliveIdleTmInSec);
	p_tConnectTO ACCESS ADR(tConnectTO);
	p_sMsgWr ACCESS ADR(sMsgWr);
	p_diStartCode1 ACCESS ADR(diStartCode1);
	p_diStartCode2 ACCESS ADR(diStartCode2);
	p_diEndCode1 ACCESS ADR(diEndCode1);
	p_diEndCode2 ACCESS ADR(diEndCode2);
	p_sProgNm ACCESS ADR(sProgNm);
	p_bNtSettingsLoadDone ACCESS ADR(bNtSettingsLoadDone);

END_ACTION
```

#### Act_LinkAction.st
```iecst
(** 2019-06-02 **)
ACTION Act_LinkAction:

	IF p_bRun THEN
		p_eAct ACCESS p_OpsTravLifULTopScan;
	ELSE
		p_eAct ACCESS ADR(eAct);
	END_IF

END_ACTION
```

#### Act_LinkEn.st
```iecst
(** 2019-06-02 **)
ACTION Act_LinkEn:

	//Link bPrep, bEn & bDis

END_ACTION
```

#### Act_Main.st
```iecst
(** 2019-06-07 **)
ACTION Act_Main:

	//Main
	CASE eStat OF

		TCPActIdle_0:
			IF eStatus <> Idle THEN	//Reset Data
				//Private
				fbClntConnect(bEn := FALSE);
				fbSnd(bEn := FALSE);
				fbRcv(bEn := FALSE);
				fbClose(bEn := FALSE);

				udiTCPIdent	:= 0;
				usiStep		:= 0;

				sStatTxt	:= a_sStatText[eStat];

			END_IF

			eStatus	:= Idle;

		TCPActFullWriteRead:
			IF eStatus = Idle OR eStatus = Busy THEN

				eStatus	:= Busy;

				sStatTxt	:= a_sStatText[eStat];

				CASE usiStep OF
					0:
						fbClntConnect.sClntIP		:= p_sClntIP;
						fbClntConnect.sSvrIP		:= p_sSvrIP;
						fbClntConnect.uiClntPort	:= p_uiClntPort;
						fbClntConnect.uiSvrPort		:= p_uiSvrPort;
						fbClntConnect(bEn := TRUE);

						IF fbClntConnect.udiStatus = 0 THEN
							udiTCPIdent	:= fbClntConnect.udiTCPIdent;
							usiStep	:= 1;
						ELSIF fbClntConnect.udiStatus < 65534 THEN
							eStatus	:= Error;

							IF fbClntConnect.udiStatus = 2309 THEN
								udiStatus	:= 10000;	//TCP Open Port Error While Full Write & Read
							ELSIF fbClntConnect.udiStatus = 2300 THEN
								udiStatus	:= 10001;	//Invalid Ident While Full Write & Read
							ELSIF fbClntConnect.udiStatus = 2307 THEN
								udiStatus	:= 10002;	//Setting Send Buffer Error While Full Write & Read
							ELSIF fbClntConnect.udiStatus = 2306 THEN
								udiStatus	:= 10003;	//Setting Receive Buffer Error While Full Write & Read
							ELSIF fbClntConnect.udiStatus = 2308 THEN
								udiStatus	:= 10004;	//Setting No Waiting Error While Full Write & Read
							ELSIF fbClntConnect.udiStatus = 2305 THEN
								udiStatus	:= 10005;	//Setting Keep Alive Error While Full Write & Read
							ELSIF fbClntConnect.udiStatus = 2304 THEN
								udiStatus	:= 10006;	//Setting Keep Alive Count Error While Full Write & Read
							ELSIF fbClntConnect.udiStatus = 2303 THEN
								udiStatus	:= 10007;	//Setting Keep Alive Idle Time Error While Full Write & Read
							ELSIF fbClntConnect.udiStatus = 2302 THEN
								udiStatus	:= 10008;	//Setting Keep Alive Interval Time Error While Full Write & Read
							ELSIF fbClntConnect.udiStatus = 2313 THEN
								udiStatus	:= 10009;	//Server Connection Failed While Full Write & Read
							ELSIF fbClntConnect.udiStatus = 2314 THEN
								udiStatus	:= 10010;	//Ident In Used While Full Write & Read
							ELSIF fbClntConnect.udiStatus = 2315 THEN
								udiStatus	:= 10011;	//Connect To Server Error While Full Write & Read
							ELSIF fbClntConnect.udiStatus = 2323 THEN
								udiStatus	:= 10012;	//Client Connect Time Out While Full Write & Read
							ELSIF fbClntConnect.udiStatus = 2310 THEN
								udiStatus	:= 10013;	//Closing TCP Error While Full Write & Read
							END_IF
						END_IF

					1:
						fbSnd.udiTCPIdent	:= udiTCPIdent;
						fbSnd.udiSndSize	:= LEN(p_sMsgWr);
						fbSnd.p_BffrDest	:= ADR(p_sMsgWr);
						fbSnd(bEn := TRUE);

						IF fbSnd.udiStatus = 0 THEN
							usiStep	:= 2;
						ELSIF fbSnd.udiStatus < 65534 THEN
							eStatus	:= Error;

							IF fbSnd.udiStatus = 2320 THEN
								udiStatus	:= 10014;	//TCP Retry Send Data Error While Full Write & Read
							ELSIF fbSnd.udiStatus = 2300 THEN
								udiStatus	:= 10015;	//Invalid Ident While Full Write & Read
							ELSIF fbSnd.udiStatus = 2321 THEN
								udiStatus	:= 10016;	//Opposite Closed Connection While Full Write & Read
							ELSIF fbSnd.udiStatus = 2322 THEN
								udiStatus	:= 10017;	//TCP Send Data Error While Full Write & Read
							END_IF
						END_IF

					2:
						fbRcv.udiTCPIdent	:= udiTCPIdent;
						fbRcv(bEn := TRUE);

						IF fbRcv.udiStatus = 0 THEN
							bMsgRdValid	:= TRUE;
							uiMsgRdLen	:= UDINT_TO_UINT(fbRcv.udiDataSizeRcv);

							//Start Code
							IF p_diStartCode1 <> -1 AND p_diStartCode2 <> -1 THEN

								iStartCodeLen	:= 2;
								siStartCode1	:= DINT_TO_SINT(p_diStartCode1);
								siStartCode2	:= DINT_TO_SINT(p_diStartCode2);
								memmove(ADR(sStartCode) , ADR(siStartCode1) , 1);
								memmove(ADR(sStartCode) + 1 , ADR(siStartCode2) , 1);

								iStartCodePos	:= FIND(sFullMsgRd , sStartCode);

							ELSIF p_diStartCode1 <> -1 AND p_diStartCode2 = -1 THEN

								iStartCodeLen	:= 1;
								siStartCode1	:= DINT_TO_SINT(p_diStartCode1);
								memmove(ADR(sStartCode) , ADR(siStartCode1) , 1);

								iStartCodePos	:= FIND(sFullMsgRd , sStartCode);

							ELSIF p_diStartCode1 = -1 AND p_diStartCode2 <> -1 THEN

								iStartCodeLen	:= 1;
								siStartCode2	:= DINT_TO_SINT(p_diStartCode2);
								memmove(ADR(sStartCode) , ADR(siStartCode2) , 1);

								iStartCodePos	:= FIND(sFullMsgRd , sStartCode);

							ELSIF p_diStartCode1 = -1 AND p_diStartCode2 = -1 THEN

								iStartCodeLen	:= 0;
								iStartCodePos	:= 0;

							END_IF

							//End Code
							IF p_diEndCode1 <> -1 AND p_diEndCode2 <> -1 THEN

								iEndCodeLen	:= 2;
								siEndCode1	:= DINT_TO_SINT(p_diEndCode1);
								siEndCode2	:= DINT_TO_SINT(p_diEndCode2);
								memmove(ADR(sEndCode) , ADR(siEndCode1) , 1);
								memmove(ADR(sEndCode) + 1 , ADR(siEndCode2) , 1);

								iEndCodePos	:= FIND(sFullMsgRd , sEndCode);

							ELSIF p_diEndCode1 <> -1 AND p_diEndCode2 = -1 THEN

								iEndCodeLen	:= 1;
								siEndCode1	:= DINT_TO_SINT(p_diEndCode1);
								memmove(ADR(sEndCode) , ADR(siEndCode1) , 1);

								iEndCodePos	:= FIND(sFullMsgRd , sEndCode);

							ELSIF p_diEndCode1 = -1 AND p_diEndCode2 <> -1 THEN

								iEndCodeLen	:= 1;
								siEndCode2	:= DINT_TO_SINT(p_diEndCode2);
								memmove(ADR(sEndCode) , ADR(siEndCode2) , 1);

								iEndCodePos	:= FIND(sFullMsgRd , sEndCode);

							ELSIF p_diEndCode1 = -1 AND p_diEndCode2 = -1 THEN

								iEndCodeLen	:= 0;
								iEndCodePos	:= 0;

							END_IF

							IF iStartCodePos = 0 THEN
								sMsgRd	:= '';
							ELSIF iEndCodePos = 0 THEN
								sMsgRd	:= RIGHT(sFullMsgRd , (LEN(sFullMsgRd) - (iStartCodePos + iStartCodeLen - 1)));
							ELSIF iEndCodePos <> 0 THEN
								sMsgRd	:= MID(sFullMsgRd , iEndCodePos - iStartCodePos - iStartCodeLen , iStartCodePos + iStartCodeLen);
							END_IF

							usiStep	:= 3;
						ELSIF fbRcv.udiStatus = 2317 THEN
							bMsgRdValid	:= FALSE;
							uiMsgRdLen	:= 0;

							usiStep		:= 3;
						ELSIF fbRcv.udiStatus < 65534 THEN
							eStatus	:= Error;

							IF fbRcv.udiStatus = 2316 THEN
								udiStatus	:= 10018;	//Data Receive Length Is Zero Due To Opposite Closed Connection While TCP Receiving Data While Full Write & Read
							ELSIF fbRcv.udiStatus = 2300 THEN
								udiStatus	:= 10019;	//Invalid Ident While Full Write & Read
							ELSIF fbRcv.udiStatus = 2318 THEN
								udiStatus	:= 10020;	//Opposite Closed Connection While Full Write & Read
							ELSIF fbRcv.udiStatus = 2319 THEN
								udiStatus	:= 10021;	//TCP Receive Data Error While Full Write & Read
							END_IF
						END_IF

					3:
						fbClose.udiTCPIdent	:= udiTCPIdent;
						fbClose(bEn := TRUE);

						IF fbClose.udiStatus = 0 THEN
							eStatus	:= Done;
						ELSIF fbClose.udiStatus < 65534 THEN
							eStatus	:= Error;

							IF fbClose.udiStatus = 2300 THEN
								udiStatus	:= 10022;	//Invalid Ident While Full Write & Read
							ELSIF fbClose.udiStatus = 2310 THEN
								udiStatus	:= 10023;	//Closing TCP Error While Full Write & Read
							END_IF
						END_IF

				END_CASE

			END_IF

		TCPActFullWriteReadUntilValid:
			IF eStatus = Idle OR eStatus = Busy THEN

				eStatus	:= Busy;

				sStatTxt	:= a_sStatText[eStat];

				CASE usiStep OF
					0:
						fbClntConnect.sClntIP		:= p_sClntIP;
						fbClntConnect.sSvrIP		:= p_sSvrIP;
						fbClntConnect.uiClntPort	:= p_uiClntPort;
						fbClntConnect.uiSvrPort		:= p_uiSvrPort;
						fbClntConnect(bEn := TRUE);

						IF fbClntConnect.udiStatus = 0 THEN
							udiTCPIdent	:= fbClntConnect.udiTCPIdent;
							udiTCPIdent1:= fbClntConnect.udiTCPIdent;

							usiStep	:= 1;
						ELSIF fbClntConnect.udiStatus < 65534 THEN
							eStatus	:= Error;

							IF fbClntConnect.udiStatus = 2309 THEN
								udiStatus	:= 10024;	//TCP Open Port Error While Full Write & Read Until Valid
							ELSIF fbClntConnect.udiStatus = 2300 THEN
								udiStatus	:= 10025;	//Invalid Ident While Full Write & Read Until Valid
							ELSIF fbClntConnect.udiStatus = 2307 THEN
								udiStatus	:= 10026;	//Setting Send Buffer Error While Full Write & Read Until Valid
							ELSIF fbClntConnect.udiStatus = 2306 THEN
								udiStatus	:= 10027;	//Setting Receive Buffer Error While Full Write & Read Until Valid
							ELSIF fbClntConnect.udiStatus = 2308 THEN
								udiStatus	:= 10028;	//Setting No Waiting Error While Full Write & Read Until Valid
							ELSIF fbClntConnect.udiStatus = 2305 THEN
								udiStatus	:= 10029;	//Setting Keep Alive Error While Full Write & Read Until Valid
							ELSIF fbClntConnect.udiStatus = 2304 THEN
								udiStatus	:= 10030;	//Setting Keep Alive Count Error While Full Write & Read Until Valid
							ELSIF fbClntConnect.udiStatus = 2303 THEN
								udiStatus	:= 10031;	//Setting Keep Alive Idle Time Error While Full Write & Read Until Valid
							ELSIF fbClntConnect.udiStatus = 2302 THEN
								udiStatus	:= 10032;	//Setting Keep Alive Interval Time Error While Full Write & Read Until Valid
							ELSIF fbClntConnect.udiStatus = 2313 THEN
								udiStatus	:= 10033;	//Server Connection Failed While Full Write & Read Until Valid
							ELSIF fbClntConnect.udiStatus = 2314 THEN
								udiStatus	:= 10034;	//Ident In Used While Full Write & Read Until Valid
							ELSIF fbClntConnect.udiStatus = 2315 THEN
								udiStatus	:= 10035;	//Connect To Server Error While Full Write & Read Until Valid
							ELSIF fbClntConnect.udiStatus = 2323 THEN
								udiStatus	:= 10036;	//Client Connect Time Out While Full Write & Read Until Valid
							ELSIF fbClntConnect.udiStatus = 2310 THEN
								udiStatus	:= 10037;	//Closing TCP Error While Full Write & Read Until Valid
							END_IF
						END_IF

					1:
						fbSnd.udiTCPIdent	:= udiTCPIdent;
						fbSnd.udiSndSize	:= LEN(p_sMsgWr);
						fbSnd.p_BffrDest	:= ADR(p_sMsgWr);

						fbSnd(bEn := TRUE);

						IF fbSnd.udiStatus = 0 THEN
							fbSnd(bEn := FALSE);
							usiStep	:= 2;
						ELSIF fbSnd.udiStatus < 65534 THEN

							fbClose.udiTCPIdent	:= udiTCPIdent;
							fbClose(bEn := TRUE);

							IF fbClose.udiStatus = 0 THEN
								fbSnd(bEn := FALSE);

								eStatus	:= Error;

								IF fbSnd.udiStatus = 2320 THEN
									udiStatus	:= 10038;	//TCP Retry Send Data Error While Full Write & Read Until Valid
								ELSIF fbSnd.udiStatus = 2300 THEN
									udiStatus	:= 10039;	//Invalid Ident While Full Write & Read Until Valid
								ELSIF fbSnd.udiStatus = 2321 THEN
									udiStatus	:= 10040;	//Opposite Closed Connection While Full Write & Read Until Valid
								ELSIF fbSnd.udiStatus = 2322 THEN
									udiStatus	:= 10041;	//TCP Send Data Error While Full Write & Read Until Valid
								END_IF
							END_IF

						END_IF

					2:
						fbRcv.udiTCPIdent	:= udiTCPIdent;
						fbRcv(bEn := TRUE);

						IF fbRcv.udiStatus = 0 THEN
							fbRcv(bEn := FALSE);
							bMsgRdValid	:= TRUE;
							uiMsgRdLen	:= UDINT_TO_UINT(fbRcv.udiDataSizeRcv);

							//Start Code
							IF p_diStartCode1 <> -1 AND p_diStartCode2 <> -1 THEN

								iStartCodeLen	:= 2;
								siStartCode1	:= DINT_TO_SINT(p_diStartCode1);
								siStartCode2	:= DINT_TO_SINT(p_diStartCode2);
								memmove(ADR(sStartCode) , ADR(siStartCode1) , 1);
								memmove(ADR(sStartCode) + 1 , ADR(siStartCode2) , 1);

								iStartCodePos	:= FIND(sFullMsgRd , sStartCode);

							ELSIF p_diStartCode1 <> -1 AND p_diStartCode2 = -1 THEN

								iStartCodeLen	:= 1;
								siStartCode1	:= DINT_TO_SINT(p_diStartCode1);
								memmove(ADR(sStartCode) , ADR(siStartCode1) , 1);

								iStartCodePos	:= FIND(sFullMsgRd , sStartCode);

							ELSIF p_diStartCode1 = -1 AND p_diStartCode2 <> -1 THEN

								iStartCodeLen	:= 1;
								siStartCode2	:= DINT_TO_SINT(p_diStartCode2);
								memmove(ADR(sStartCode) , ADR(siStartCode2) , 1);

								iStartCodePos	:= FIND(sFullMsgRd , sStartCode);

							ELSIF p_diStartCode1 = -1 AND p_diStartCode2 = -1 THEN

								iStartCodeLen	:= 0;
								iStartCodePos	:= 0;

							END_IF

							//End Code
							IF p_diEndCode1 <> -1 AND p_diEndCode2 <> -1 THEN

								iEndCodeLen	:= 2;
								siEndCode1	:= DINT_TO_SINT(p_diEndCode1);
								siEndCode2	:= DINT_TO_SINT(p_diEndCode2);
								memmove(ADR(sEndCode) , ADR(siEndCode1) , 1);
								memmove(ADR(sEndCode) + 1 , ADR(siEndCode2) , 1);

								iEndCodePos	:= FIND(sFullMsgRd , sEndCode);

							ELSIF p_diEndCode1 <> -1 AND p_diEndCode2 = -1 THEN

								iEndCodeLen	:= 1;
								siEndCode1	:= DINT_TO_SINT(p_diEndCode1);
								memmove(ADR(sEndCode) , ADR(siEndCode1) , 1);

								iEndCodePos	:= FIND(sFullMsgRd , sEndCode);

							ELSIF p_diEndCode1 = -1 AND p_diEndCode2 <> -1 THEN

								iEndCodeLen	:= 1;
								siEndCode2	:= DINT_TO_SINT(p_diEndCode2);
								memmove(ADR(sEndCode) , ADR(siEndCode2) , 1);

								iEndCodePos	:= FIND(sFullMsgRd , sEndCode);

							ELSIF p_diEndCode1 = -1 AND p_diEndCode2 = -1 THEN

								iEndCodeLen	:= 0;
								iEndCodePos	:= 0;

							END_IF

							IF iStartCodePos = 0 THEN
								sMsgRd	:= '';
							ELSIF iEndCodePos = 0 THEN
								sMsgRd	:= RIGHT(sFullMsgRd , (LEN(sFullMsgRd) - (iStartCodePos + iStartCodeLen - 1)));
							ELSIF iEndCodePos <> 0 THEN
								sMsgRd	:= MID(sFullMsgRd , iEndCodePos - iStartCodePos - iStartCodeLen , iStartCodePos + iStartCodeLen);
							END_IF

							IF p_usiTravLifScanCntr = usiScanCntr THEN //number of scan
								usiStep	:= 3;
							ELSE
								usiScanCntr := usiScanCntr +1;
								eStatus := Done;
							END_IF

						ELSIF fbRcv.udiStatus = 2317 THEN
							fbRcv(bEn := FALSE);
						ELSIF fbRcv.udiStatus < 65534 THEN
							eStatus	:= Error;

							IF fbRcv.udiStatus = 2316 THEN
								udiStatus	:= 10042;	//Data Receive Length Is Zero Due To Opposite Closed Connection While TCP Receiving Data While Full Write & Read Until Valid
							ELSIF fbRcv.udiStatus = 2300 THEN
								udiStatus	:= 10043;	//Invalid Ident While Full Write & Read Until Valid
							ELSIF fbRcv.udiStatus = 2318 THEN
								bRstConnection := TRUE;
								udiStatus	:= 10044;	//Opposite Closed Connection While Full Write & Read Until Valid
							ELSIF fbRcv.udiStatus = 2319 THEN
								udiStatus	:= 10045;	//TCP Receive Data Error While Full Write & Read Until Valid
							END_IF
						END_IF

					3:
						fbClose.udiTCPIdent	:= udiTCPIdent;
						fbClose(bEn := TRUE);

						IF fbClose.udiStatus = 0 THEN
							udiTCPIdent := 0;
							eStatus	:= Done;
						ELSIF fbClose.udiStatus < 65534 THEN
							eStatus	:= Error;

							IF fbClose.udiStatus = 2300 THEN
								udiStatus	:= 10046;	//Invalid Ident While Full Write & Read Until Valid
							ELSIF fbClose.udiStatus = 2310 THEN
								udiStatus	:= 10047;	//Closing TCP Error While Full Write & Read Until Valid
							END_IF
						END_IF

				END_CASE

			END_IF

		TCPActDebug :
			IF eStatus = Idle OR eStatus = Busy THEN

				eStatus	:= Busy;

				sStatTxt	:= a_sStatText[eStat];

				CASE usiStep OF
					0:
						fbClntConnect.sClntIP		:= p_sClntIP;
						fbClntConnect.sSvrIP		:= p_sSvrIP;
						fbClntConnect.uiClntPort	:= p_uiClntPort;
						fbClntConnect.uiSvrPort		:= p_uiSvrPort;
						fbClntConnect(bEn := TRUE);

						IF fbClntConnect.udiStatus = 0 THEN
							udiTCPIdent	:= fbClntConnect.udiTCPIdent;

						//	usiStep	:= 1;
						ELSIF fbClntConnect.udiStatus < 65534 THEN
							eStatus	:= Error;

							IF fbClntConnect.udiStatus = 2309 THEN
								udiStatus	:= 10024;	//TCP Open Port Error While Full Write & Read Until Valid
							ELSIF fbClntConnect.udiStatus = 2300 THEN
								udiStatus	:= 10025;	//Invalid Ident While Full Write & Read Until Valid
							ELSIF fbClntConnect.udiStatus = 2307 THEN
								udiStatus	:= 10026;	//Setting Send Buffer Error While Full Write & Read Until Valid
							ELSIF fbClntConnect.udiStatus = 2306 THEN
								udiStatus	:= 10027;	//Setting Receive Buffer Error While Full Write & Read Until Valid
							ELSIF fbClntConnect.udiStatus = 2308 THEN
								udiStatus	:= 10028;	//Setting No Waiting Error While Full Write & Read Until Valid
							ELSIF fbClntConnect.udiStatus = 2305 THEN
								udiStatus	:= 10029;	//Setting Keep Alive Error While Full Write & Read Until Valid
							ELSIF fbClntConnect.udiStatus = 2304 THEN
								udiStatus	:= 10030;	//Setting Keep Alive Count Error While Full Write & Read Until Valid
							ELSIF fbClntConnect.udiStatus = 2303 THEN
								udiStatus	:= 10031;	//Setting Keep Alive Idle Time Error While Full Write & Read Until Valid
							ELSIF fbClntConnect.udiStatus = 2302 THEN
								udiStatus	:= 10032;	//Setting Keep Alive Interval Time Error While Full Write & Read Until Valid
							ELSIF fbClntConnect.udiStatus = 2313 THEN
								udiStatus	:= 10033;	//Server Connection Failed While Full Write & Read Until Valid
							ELSIF fbClntConnect.udiStatus = 2314 THEN
								udiStatus	:= 10034;	//Ident In Used While Full Write & Read Until Valid
							ELSIF fbClntConnect.udiStatus = 2315 THEN
								udiStatus	:= 10035;	//Connect To Server Error While Full Write & Read Until Valid
							ELSIF fbClntConnect.udiStatus = 2323 THEN
								udiStatus	:= 10036;	//Client Connect Time Out While Full Write & Read Until Valid
							ELSIF fbClntConnect.udiStatus = 2310 THEN
								udiStatus	:= 10037;	//Closing TCP Error While Full Write & Read Until Valid
							END_IF
						END_IF

					1:
						fbSnd.udiTCPIdent	:= udiTCPIdent;
						fbSnd.udiSndSize	:= LEN(p_sMsgWr);
						fbSnd.p_BffrDest	:= ADR(p_sMsgWr);
						fbSnd(bEn := TRUE);

						IF fbSnd.udiStatus = 0 THEN
						//	usiStep	:= 2;
						ELSIF fbSnd.udiStatus < 65534 THEN
							eStatus	:= Error;

							IF fbSnd.udiStatus = 2320 THEN
								udiStatus	:= 10038;	//TCP Retry Send Data Error While Full Write & Read Until Valid
							ELSIF fbSnd.udiStatus = 2300 THEN
								udiStatus	:= 10039;	//Invalid Ident While Full Write & Read Until Valid
							ELSIF fbSnd.udiStatus = 2321 THEN
								udiStatus	:= 10040;	//Opposite Closed Connection While Full Write & Read Until Valid
							ELSIF fbSnd.udiStatus = 2322 THEN
								udiStatus	:= 10041;	//TCP Send Data Error While Full Write & Read Until Valid
							END_IF
						END_IF

					2:
						fbRcv.udiTCPIdent	:= udiTCPIdent;
						fbRcv(bEn := TRUE);

						IF fbRcv.udiStatus = 0 THEN
							bMsgRdValid	:= TRUE;
							uiMsgRdLen	:= UDINT_TO_UINT(fbRcv.udiDataSizeRcv);

							sMsgRd	:= MID(sFullMsgRd , iEndCodePos - iStartCodePos - iStartCodeLen , iStartCodePos + iStartCodeLen);

						//	usiStep	:= 3;
						ELSIF fbRcv.udiStatus = 2317 THEN
							fbRcv(bEn := FALSE);
						ELSIF fbRcv.udiStatus < 65534 THEN
							eStatus	:= Error;

							IF fbRcv.udiStatus = 2316 THEN
								udiStatus	:= 10042;	//Data Receive Length Is Zero Due To Opposite Closed Connection While TCP Receiving Data While Full Write & Read Until Valid
							ELSIF fbRcv.udiStatus = 2300 THEN
								udiStatus	:= 10043;	//Invalid Ident While Full Write & Read Until Valid
							ELSIF fbRcv.udiStatus = 2318 THEN
								udiStatus	:= 10044;	//Opposite Closed Connection While Full Write & Read Until Valid
							ELSIF fbRcv.udiStatus = 2319 THEN
								udiStatus	:= 10045;	//TCP Receive Data Error While Full Write & Read Until Valid
							END_IF
						END_IF

					3:
						fbClose.udiTCPIdent	:= udiTCPIdent;
						fbClose(bEn := TRUE);

						IF fbClose.udiStatus = 0 THEN
						//	eStatus	:= Done;
						ELSIF fbClose.udiStatus < 65534 THEN
							eStatus	:= Error;

							IF fbClose.udiStatus = 2300 THEN
								udiStatus	:= 10046;	//Invalid Ident While Full Write & Read Until Valid
							ELSIF fbClose.udiStatus = 2310 THEN
								udiStatus	:= 10047;	//Closing TCP Error While Full Write & Read Until Valid
							END_IF
						END_IF

				END_CASE
			END_IF
	END_CASE

END_ACTION
```

#### Act_RstErr.st
```iecst
(** 2019-06-02 **)
ACTION Act_RstErr:

	IF p_udiRstErr <> udiRstErrOld THEN
		bRstErr			:= TRUE;
		udiRstErrOld	:= p_udiRstErr;
	ELSE
		bRstErr			:= FALSE;
	END_IF

	IF (bRstConnection AND eStat = TCPActIdle_0) OR ((bRstErr OR fbClose.bEn =TRUE) AND udiTCPIdent1 <> 0 AND eStat = TCPActIdle_0 )THEN
		fbClose.udiTCPIdent	:= udiTCPIdent1;
		fbClose(bEn := TRUE);

		IF fbClose.udiStatus = 0 THEN
			udiTCPIdent	:= 0;
			fbClose(bEn := FALSE);
			bRstConnection := FALSE;
			udiTCPIdent1 := 0;
		ELSIF fbClose.udiStatus < 65534 THEN
			udiTCPIdent	:= 0;
			eStatus	:= Error;

			IF fbClose.udiStatus = 2300 THEN
				udiStatus	:= 10146;	//Invalid Ident While Closing TCP
			ELSIF fbClose.udiStatus = 2310 THEN
				udiStatus	:= 10147;	//Closing TCP Error
			ELSE
				udiStatus	:= fbClose.udiStatus;
			END_IF

		END_IF
	END_IF

END_ACTION
```

#### Cyclic.st
```iecst
(** 2019-06-02 **)
PROGRAM _CYCLIC

	IF bInitDone = FALSE THEN
		bInitDone	:= TRUE;

		Act_InitLocal;
		Act_InitGlobal;

	ELSIF bInitialDone = FALSE THEN
		IF p_bNtSettingsLoadDone = TRUE THEN
			bInitialDone	:= TRUE;

			Act_Initial;
		END_IF

	ELSE

		Act_RstErr;
		Act_LinkAction;
		Act_Action;
		Act_LinkEn;

		IF (p_bPrep = TRUE) AND (p_bEn = TRUE) AND (p_bDis = FALSE) THEN
			Act_Link;
			Act_Background;
			Act_Main;
		ELSE
			IF eStat <> TCPActIdle_0 THEN
				eStatus	:= Done;
			ELSE
				eStatus	:= Idle;
			END_IF
		END_IF

		Act_Alarm;

	END_IF

END_PROGRAM
```

#### Init.st
```iecst
(** 2019-06-02 **)
PROGRAM _INIT

	(* Always Change If Project Change *)

	//Pass Address To Global Address For External Use
	//Action, State & Status
	p_TCPTopStat		:= ADR(eStat);
	p_TCPTopStatus		:= ADR(eStatus);
	p_TCPTopStatTxt		:= ADR(sStatTxt);

	//Alarm
	p_TCPTopAlmData		:= ADR(tyAlmData);

	//Output
	p_TCPTopFullMsgRd	:= ADR(sFullMsgRd);
	p_TCPTopMsgRd		:= ADR(sMsgRd);
	p_TCPTopMsgRdValid	:= ADR(bMsgRdValid);
	p_TCPTopMsgRdLen	:= ADR(uiMsgRdLen);

	(* Always Change If Project Change *)

END_PROGRAM
```

### TCPBtm.var - Change By Project
```iecst
(*2019-06-02*)
(**)
(*Constant*)
(**)
(*Action & State & Status*)
VAR
	p_TCPBtmStat : UDINT;
	p_TCPBtmStatus : UDINT;
	p_TCPBtmStatTxt : UDINT;
END_VAR
(**)
(*Alarm*)
VAR
	p_TCPBtmAlmData : UDINT;
END_VAR
(**)
(*Output*)
VAR
	p_TCPBtmFullMsgRd : UDINT;
	p_TCPBtmMsgRd : UDINT;
	p_TCPBtmMsgRdValid : UDINT;
	p_TCPBtmMsgRdLen : UDINT;
END_VAR
```

### Program Logical/TCP/TCPBtm (IEC) - 1.00.0 - NtRecipe v5.00.0 , NtFileIO v5.00.0

#### Local.var
```iecst
(*2019-06-07*)
(**)
(*Local Action, State & Status*)
VAR
	eAct : eTCPAction1 := TCPActIdle_0;
	eStat : eTCPAction1 := TCPActIdle_0;
	eStatus : eFBStatus := Idle;
	udiStatus : UDINT := 0;
	sStatTxt : STRING[200] := '';
	a_sStatText : ARRAY[0..50] OF STRING[200] := ['Idling','TCP Write Then Read','TCP Write Then Read Until Valid',48('')];
END_VAR
(**)
(*Local Alarm*)
VAR
	tyAlmData : tyAlmDat;
	a_tyAlmText : ARRAY[10000..10099] OF tyAlmTxt := [(sAlmText:='TCP Open Port Error While Full Write & Read',sRcyText:='Pleae Contact Nutek For Future Possible Solution'),(sAlmText:='Invalid Ident While Full Write & Read',sRcyText:='Pleae Contact Nutek For Future Possible Solution'),(sAlmText:='Setting Send Buffer Error While Full Write & Read',sRcyText:='Pleae Contact Nutek For Future Possible Solution'),(sAlmText:='Setting Receive Buffer Error While Full Write & Read',sRcyText:='Pleae Contact Nutek For Future Possible Solution'),(sAlmText:='Setting No Waiting Error While Full Write & Read',sRcyText:='Pleae Contact Nutek For Future Possible Solution'),(sAlmText:='Setting Keep Alive Error While Full Write & Read',sRcyText:='Pleae Contact Nutek For Future Possible Solution'),(sAlmText:='Setting Keep Alive Count Error While Full Write & Read',sRcyText:='Pleae Contact Nutek For Future Possible Solution'),(sAlmText:='Setting Keep Alive Idle Time Error While Full Write & Read',sRcyText:='Pleae Contact Nutek For Future Possible Solution'),(sAlmText:='Setting Keep Alive Interval Time Error While Full Write & Read',sRcyText:='Pleae Contact Nutek For Future Possible Solution'),(sAlmText:='Server Connection Failed While Full Write & Read',sRcyText:='Check Whether Server Connection Is Valid'),(sAlmText:='Ident In Used While Full Write & Read',sRcyText:='Pleae Contact Nutek For Future Possible Solution'),(sAlmText:='Connect To Server Error While Full Write & Read',sRcyText:='Check Whether Server Connection Is Valid'),(sAlmText:='Client Connect Time Out While Full Write & Read',sRcyText:='Check Whether Server Connection Is Valid'),(sAlmText:='Closing TCP Error While Full Write & Read',sRcyText:='Pleae Contact Nutek For Future Possible Solution'),(sAlmText:='TCP Retry Send Data Error While Full Write & Read',sRcyText:='Pleae Contact Nutek For Future Possible Solution'),(sAlmText:='Invalid Ident While Full Write & Read',sRcyText:='Pleae Contact Nutek For Future Possible Solution'),(sAlmText:='Opposite Closed Connection While Full Write & Read',sRcyText:='Check Whether Server Connection Is Valid'),(sAlmText:='TCP Send Data Error While Full Write & Read',sRcyText:='Pleae Contact Nutek For Future Possible Solution'),(sAlmText:='Data Receive Length Is Zero Due To Opposite Closed Connection While TCP Receiving Data While Full Write & Read',sRcyText:='Check Whether Server Connection Is Valid'),(sAlmText:='Invalid Ident While Full Write & Read',sRcyText:='Pleae Contact Nutek For Future Possible Solution'),(sAlmText:='Opposite Closed Connection While Full Write & Read',sRcyText:='Check Whether Server Connection Is Valid'),(sAlmText:='TCP Receive Data Error While Full Write & Read',sRcyText:='Pleae Contact Nutek For Future Possible Solution'),(sAlmText:='Invalid Ident While Full Write & Read',sRcyText:='Pleae Contact Nutek For Future Possible Solution'),(sAlmText:='Closing TCP Error While Full Write & Read',sRcyText:='Pleae Contact Nutek For Future Possible Solution'),(sAlmText:='TCP Open Port Error While Full Write & Read Until Valid',sRcyText:='Pleae Contact Nutek For Future Possible Solution'),(sAlmText:='Invalid Ident While Full Write & Read Until Valid',sRcyText:='Pleae Contact Nutek For Future Possible Solution'),(sAlmText:='Setting Send Buffer Error While Full Write & Read Until Valid',sRcyText:='Pleae Contact Nutek For Future Possible Solution'),(sAlmText:='Setting Receive Buffer Error While Full Write & Read Until Valid',sRcyText:='Pleae Contact Nutek For Future Possible Solution'),(sAlmText:='Setting No Waiting Error While Full Write & Read Until Valid',sRcyText:='Pleae Contact Nutek For Future Possible Solution'),(sAlmText:='Setting Keep Alive Error While Full Write & Read Until Valid',sRcyText:='Pleae Contact Nutek For Future Possible Solution'),(sAlmText:='Setting Keep Alive Count Error While Full Write & Read Until Valid',sRcyText:='Pleae Contact Nutek For Future Possible Solution'),(sAlmText:='Setting Keep Alive Idle Time Error While Full Write & Read Until Valid',sRcyText:='Pleae Contact Nutek For Future Possible Solution'),(sAlmText:='Setting Keep Alive Interval Time Error While Full Write & Read Until Valid',sRcyText:='Pleae Contact Nutek For Future Possible Solution'),(sAlmText:='Server Connection Failed While Full Write & Read Until Valid',sRcyText:='Check Whether Server Connection Is Valid'),(sAlmText:='Ident In Used While Full Write & Read Until Valid',sRcyText:='Pleae Contact Nutek For Future Possible Solution'),(sAlmText:='Connect To Server Error While Full Write & Read Until Valid',sRcyText:='Check Whether Server Connection Is Valid'),(sAlmText:='Client Connect Time Out While Full Write & Read Until Valid',sRcyText:='Check Whether Server Connection Is Valid'),(sAlmText:='Closing TCP Error While Full Write & Read Until Valid',sRcyText:='Pleae Contact Nutek For Future Possible Solution'),(sAlmText:='TCP Retry Send Data Error While Full Write & Read Until Valid',sRcyText:='Pleae Contact Nutek For Future Possible Solution'),(sAlmText:='Invalid Ident While Full Write & Read Until Valid',sRcyText:='Pleae Contact Nutek For Future Possible Solution'),(sAlmText:='Opposite Closed Connection While Full Write & Read Until Valid',sRcyText:='Check Whether Server Connection Is Valid'),(sAlmText:='TCP Send Data Error While Full Write & Read Until Valid',sRcyText:='Pleae Contact Nutek For Future Possible Solution'),(sAlmText:='Data Receive Length Is Zero Due To Opposite Closed Connection While TCP Receiving Data While Full Write & Read Until Valid',sRcyText:='Check Whether Server Connection Is Valid'),(sAlmText:='Invalid Ident While Full Write & Read Until Valid',sRcyText:='Pleae Contact Nutek For Future Possible Solution'),(sAlmText:='Opposite Closed Connection While Full Write & Read Until Valid',sRcyText:='Check Whether Server Connection Is Valid'),(sAlmText:='TCP Receive Data Error While Full Write & Read Until Valid',sRcyText:='Pleae Contact Nutek For Future Possible Solution'),(sAlmText:='Invalid Ident While Full Write & Read Until Valid',sRcyText:='Pleae Contact Nutek For Future Possible Solution'),(sAlmText:='Closing TCP Error While Full Write & Read Until Valid',sRcyText:='Pleae Contact Nutek For Future Possible Solution'),52(0)];
END_VAR
(**)
(*Local Output*)
VAR
	sFullMsgRd : STRING[80];
	sMsgRd : STRING[80];
	bMsgRdValid : BOOL;
	uiMsgRdLen : UINT;
END_VAR
(**)
(*Local Input*)
VAR
	udiRstErr : UDINT := 0;
	bPrep : BOOL := TRUE;
	bEn : BOOL := TRUE;
	bDis : BOOL := FALSE;
	bRun : BOOL := FALSE;
	sClntIP : STRING[15];
	sSvrIP : STRING[15];
	uiClntPort : UINT;
	uiSvrPort : UINT;
	udiSndBffrSize : UDINT := 65536;
	udiRcvBffrSize : UDINT := 65536;
	udiAliveIdleTmInSec : UDINT := 10;
	tConnectTO : TIME := T#30s;
	sMsgWr : STRING[80] := 'T'; (*trigger scanner*)
	diStartCode1 : DINT := -1;
	diStartCode2 : DINT := -1;
	diEndCode1 : DINT := -1;
	diEndCode2 : DINT := -1;
	sProgNm : STRING[15] := 'TCPTop';
	bNtSettingsLoadDone : BOOL := TRUE;
END_VAR
(**)
(*Local*)
VAR
	bRstErr : BOOL;
	udiRstErrOld : UDINT;
	bInitDone : BOOL;
	bInitialDone : BOOL;
	fbClntConnect : fbTCPClntConnect;
	fbSnd : fbTCPSnd;
	fbRcv : fbTCPRcv;
	fbClose : fbTCPClose;
	udiTCPIdent : UDINT;
	udiTCPIdent1 : UDINT;
	usiStep : USINT;
	iStartCodeLen : INT;
	siStartCode1 : SINT;
	siStartCode2 : SINT;
	sStartCode : STRING[2];
	iStartCodePos : INT;
	iEndCodeLen : INT;
	siEndCode1 : SINT;
	siEndCode2 : SINT;
	sEndCode : STRING[2];
	iEndCodePos : INT;
	bRstConnection : BOOL;
	usiScanCntr : USINT;
	bTest : BOOL;
END_VAR
```

#### Act_Background.st
```iecst
(** 2019-06-02 **)
ACTION Act_Background:

END_ACTION
```

#### Act_InitGlobal.st
```iecst
(** 2019-06-02 **)
ACTION Act_InitGlobal:

	(* Always Change If Project Change *)

	//Pass Data To Link

	//Pass Data To Internal Use
	p_bPrep ACCESS p_NtParamProjScanPrep;
	p_bEn ACCESS p_McParamBtmScannerEn;
	p_udiRstErr ACCESS p_RstErrReset;

	p_sClntIP ACCESS p_HWInfoIPAddr;
	p_sSvrIP ACCESS p_McParamBtmScanIP;
	p_uiSvrPort ACCESS p_McParamBtmScanPort;
	p_bRun ACCESS p_OpsRun;

	p_bNtSettingsLoadDone ACCESS p_StartupNtSettingsLoadDone;
	p_usiTravLifScanCntr ACCESS p_OpsTravLifScanCntr;
	(* Always Change If Project Change *)

END_ACTION
```

#### Act_Initial.st
```iecst
(** 2019-06-02 **)
ACTION Act_Initial:

	//Initial
	sStatTxt	:= a_sStatText[eStat];

	fbClntConnect.udiSndBffrSize		:= p_udiSndBffrSize;
	fbClntConnect.udiRcvBffrSize		:= p_udiRcvBffrSize;
	fbClntConnect.udiAliveIdleTmInSec	:= p_udiAliveIdleTmInSec;
	fbClntConnect.tConnectTO			:= p_tConnectTO;
	fbClntConnect(bEn := FALSE);

	fbSnd(bEn := FALSE);

	fbRcv.udiBffrSize	:= SIZEOF(sFullMsgRd);
	fbRcv.p_BffrDest	:= ADR(sFullMsgRd);
	fbRcv(bEn := FALSE);

	fbClose(bEn := FALSE);

END_ACTION
```

#### Act_Link.st
```iecst
(** 2019-06-02 **)
ACTION Act_Link:

	IF EDGEPOS(bTest ) THEN
		iStartCodeLen	:= 2;
		siStartCode1	:= DINT_TO_SINT(p_diStartCode1);
		siStartCode2	:= DINT_TO_SINT(p_diStartCode2);
		memmove(ADR(sStartCode) , ADR(siStartCode1) , 1);
		memmove(ADR(sStartCode) + 1 , ADR(siStartCode2) , 1);

		iStartCodePos	:= FIND(sFullMsgRd , sStartCode);
	END_IF

END_ACTION
```

#### Act_LinkAction.st
```iecst
(** 2019-06-02 **)
ACTION Act_LinkAction:

	IF p_bRun THEN
		p_eAct ACCESS p_OpsTravLifULBtmScan;
	ELSE
		p_eAct ACCESS ADR(eAct);
	END_IF

END_ACTION
```
